	// Check buffer alarm
	IF fbMFCS_Channel[E_MFCS_Channel.AM].M_BufferLevelAlarm() THEN	
		// Set error
		F_SetError(	
			ErrorType	:= E_ErrorType.ERROR,
			ErrorParam	:= '',
			ErrorMsg	:= E_ErrorConv.AM_BUFFER_OVERFLOW,
			ErrorData	:= SubsystemData.ErrorData.ErrorDataSet[7]);
			
	// Check buffer warning
	ELSIF fbMFCS_Channel[E_MFCS_Channel.AM].M_BufferLevelWarning() AND
	      SubsystemData.ErrorData.ErrorDataSet[7].ErrorType <> E_ErrorType.ERROR THEN
		// Set error
		F_SetError(	
			ErrorType	:= E_ErrorType.WARNING,
			ErrorParam	:= '',
			ErrorMsg	:= E_ErrorConv.AM_BUFFER_OVERFLOW,
			ErrorData	:= SubsystemData.ErrorData.ErrorDataSet[7]);
	ELSE
		// Reset error
		F_ResetError(Reset := TRUE, ErrorData := SubsystemData.ErrorData.ErrorDataSet[7]);
		
	END_IF
ELSE
	// Reset error
	F_ResetError(Reset := TRUE, ErrorData := SubsystemData.ErrorData.ErrorDataSet[6]);
	F_ResetError(Reset := TRUE, ErrorData := SubsystemData.ErrorData.ErrorDataSet[7]);
	
	// Reset command to stop
	StopAllGroups := FALSE;
END_IF

(**************************************************************************************
   SPOC Connection
***************************************************************************************)
// If SPOC is configured
IF Settings.SPOC_Exists THEN
	
	// If SPOC is not connected
	IF NOT fbMFCS_Channel[E_MFCS_Channel.SPOC].M_IsConnected() THEN
		// Set error
		F_SetError(	
			ErrorType	:= E_ErrorType.ERROR,
			ErrorParam	:= '',
			ErrorMsg	:= E_ErrorConv.CONNECTION_ERROR_TO_SPOC,
			ErrorData	:= SubsystemData.ErrorData.ErrorDataSet[8]);
	ELSE
		// Reset error
		F_ResetError(Reset := TRUE,ErrorData := SubsystemData.ErrorData.ErrorDataSet[8]);
	END_IF
ELSE
	// Reset error
	F_ResetError(Reset := TRUE,ErrorData := SubsystemData.ErrorData.ErrorDataSet[8]);
END_IF
END_ACTION

ACTION A_OutputMapping:
(**************************************************************************************
 * 	NAME		A_OutputMapping
 * 	FUNCTION	Output mapping
 **************************************************************************************)

 
 
(**************************************************************************************************************
   Outputs
***************************************************************************************************************)
SubsystemInterface.Out.MasterSpeed := SubsystemInterface.In.MasterSpeed;
END_ACTION

ACTION A_SlaveDeviceSupervision:
(**************************************************************************************
 * 	NAME		A_SlaveDeviceSupervision
 * 	FUNCTION	Check connected EtherCAT Slaves for diagnostic reasons
 *
 *				0x___1 = Slave in 'INIT' state
 *	 			0x___2 = Slave in 'PREOP' state
 *				0x___3 = Slave in 'BOOT' state
 *				0x___4 = Slave in 'SAFEOP' state
 *				0x___8 = Slave in 'OP' state
 *				0x001_ = Slave signals error
 *				0x002_ = Invalid vendorId, productCode... read
 *				0x004_ = Initialization error occurred
 *				0x008_ = Slave disabled
 *				0x010_ = Slave not present
 *				0x020_ = Slave signals link error
 *				0x040_ = Slave signals missing link
 *				0x080_ = Slave signals unexpected link
 *				0x100_ = Communication port A
 *				0x200_ = Communication port B
 *				0x400_ = Communication port C
 *				0x800_ = Communication port D
 *
 **************************************************************************************)
 
// Check all device slaves 
FOR Idx := 1 TO NUMBERS_OF_ETHERCAT_SLAVE_DIAG DO
	// If state is >16 and state has changed
	IF Inputs.DeviceState[Idx] >= 16 AND Inputs.DeviceState[Idx] <> EtherCatSupervision[Idx].DeviceState THEN
		// Update event list
		EtherCatSupervision[Idx].EventDateTime 			:= TimeStampDT;
		EtherCatSupervision[Idx].Error 					:= TRUE;
		EtherCatSupervision[Idx].LastDeviceState		:= EtherCatSupervision[Idx].DeviceState;
		EtherCatSupervision[Idx].DeviceState			:= Inputs.DeviceState[Idx];
		
		// Print debug
		DebugMsg := CONCAT('EtherCAT-Device Error, Device: ', INT_TO_STRING(Idx));
		DebugMsg := CONCAT(DebugMsg, ' Last Device state: ');
		DebugMsg := CONCAT(DebugMsg, UINT_TO_STRING(EtherCatSupervision[Idx].LastDeviceState));
		DebugMsg := CONCAT(DebugMsg, ' Device state: ');
		DebugMsg := CONCAT(DebugMsg, UINT_TO_STRING(EtherCatSupervision[Idx].DeviceState));
		DebugMsg := CONCAT(DebugMsg, ' Active: ');
		DebugMsg := CONCAT(DebugMsg, BOOL_TO_STRING(EtherCatSupervision[Idx].Error));
		fbDebugMsg.M_SendInfoMsg(DebugMsg);
		
	// If no error is active - update table
	ELSIF Inputs.DeviceState[Idx] <> EtherCatSupervision[Idx].DeviceState THEN
		// Reset table
		EtherCatSupervision[Idx].LastDeviceState		:= EtherCatSupervision[Idx].DeviceState;
		EtherCatSupervision[Idx].DeviceState			:= Inputs.DeviceState[Idx];
		EtherCatSupervision[Idx].Error	 				:= FALSE;
		
		// Print debug
		DebugMsg := CONCAT('EtherCAT-Device Error, Device: ', INT_TO_STRING(Idx));
		DebugMsg := CONCAT(DebugMsg, ' Last Device state: ');
		DebugMsg := CONCAT(DebugMsg, UINT_TO_STRING(EtherCatSupervision[Idx].LastDeviceState));
		DebugMsg := CONCAT(DebugMsg, ' Device state: ');
		DebugMsg := CONCAT(DebugMsg, UINT_TO_STRING(EtherCatSupervision[Idx].DeviceState));
		DebugMsg := CONCAT(DebugMsg, ' Active: ');
		DebugMsg := CONCAT(DebugMsg, BOOL_TO_STRING(EtherCatSupervision[Idx].Error));
		fbDebugMsg.M_SendInfoMsg(DebugMsg);
	END_IF
END_FOR
END_ACTION

ACTION A_StateControl:
(**************************************************************************************
 * 	NAME		A_StateControl
 * 	FUNCTION	State control 
 **************************************************************************************)

// Update system state
SubSystemData.OperationState.Info.SystemReady := SubSystemData.OperationState.eState = E_PositionState.STARTED;
 
// Group states
CASE SubSystemData.OperationState.eState OF
	(*******************************************************************************
	  Unknown State 
	********************************************************************************)
	E_PositionState.UNKNOWN:
		// Subsystem default state
		SubSystemData.OperationState.eLastState := SubSystemData.OperationState.eState;
		SubSystemData.OperationState.eState 	:= E_PositionState.STOPPED;

	(*******************************************************************************
	  Stopped
	********************************************************************************)
	E_PositionState.STOPPED:
		IF SubSystemData.ErrorData.ErrorDataSet[7].ErrorType <> E_ErrorType.ERROR AND
		   SubSystemData.ErrorData.ErrorDataSet[7].ErrorType <> E_ErrorType.WARNING THEN
		   
		   // Change state "Starting"
			SubSystemData.OperationState.eLastState := SubSystemData.OperationState.eState;
			SubSystemData.OperationState.eState := E_PositionState.STARTING;
		
			// Send status report
			ITC.Commands.StatusReport := TRUE;
		END_IF
		
	(*******************************************************************************
	  Stopping
	********************************************************************************)
	E_PositionState.STOPPING:
		fbStoppingDelayTimer(IN := TRUE, PT := Settings.tDelayStopping);
	
		// If no "AM_Buffer" error is pending
		IF SubSystemData.ErrorData.ErrorDataSet[7].ErrorType = E_ErrorType.ERROR OR 
		   fbStoppingDelayTimer.Q THEN
		   
			// Change state "Stopped"
			SubSystemData.OperationState.eLastState := SubSystemData.OperationState.eState;
			SubSystemData.OperationState.eState := E_PositionState.STOPPED;
		
			// Send status report
			ITC.Commands.StatusReport := TRUE;
			
			fbStoppingDelayTimer(IN := FALSE);
			
		// If no "AM_BUffer" warning is pending
		ELSIF SubSystemData.ErrorData.ErrorDataSet[7].ErrorType = E_ErrorType.WARNING THEN
			// Wait
			;
		ELSE
			// Start again
			SubSystemData.OperationState.eLastState := SubSystemData.OperationState.eState;
			SubSystemData.OperationState.eState := E_PositionState.STARTING;
		
			// Send status report
			ITC.Commands.StatusReport := TRUE;
		END_IF

	(*******************************************************************************
	  Starting
	********************************************************************************)
	E_PositionState.STARTING:
		// If no "AM_Buffer" error/warning is pending
		IF SubSystemData.ErrorData.ErrorDataSet[7].ErrorType = E_ErrorType.ERROR OR
   		   SubSystemData.ErrorData.ErrorDataSet[7].ErrorType = E_ErrorType.WARNING THEN
			// Change state "Stopped"
			SubSystemData.OperationState.eLastState := SubSystemData.OperationState.eState;
			SubSystemData.OperationState.eState := E_PositionState.STOPPED;
		
			// Send status report
			ITC.Commands.StatusReport := TRUE;
			
		ELSIF fbStartUpDelayTimer.Q THEN
			// Change state "Started"
			SubSystemData.OperationState.eLastState := SubSystemData.OperationState.eState;
			SubSystemData.OperationState.eState := E_PositionState.STARTED;
		
			// Send status report
			ITC.Commands.StatusReport := TRUE;
		END_IF
		
	(*******************************************************************************
	  Started (Online/active/running)
	********************************************************************************)
	E_PositionState.STARTED:
	
		// If no "AM_Buffer" error is pending
		IF SubSystemData.ErrorData.ErrorDataSet[7].ErrorType = E_ErrorType.ERROR OR
		   NOT fbStartUpDelayTimer.Q THEN
			// Change state "Stopped"
			SubSystemData.OperationState.eLastState := SubSystemData.OperationState.eState;
			SubSystemData.OperationState.eState := E_PositionState.STOPPED;
			// Send status report
			ITC.Commands.StatusReport := TRUE;
			
		// If no "AM_BUffer" warning is pending
		ELSIF SubSystemData.ErrorData.ErrorDataSet[7].ErrorType = E_ErrorType.WARNING THEN
			// Change state "Stopping"
			SubSystemData.OperationState.eLastState := SubSystemData.OperationState.eState;
			SubSystemData.OperationState.eState := E_PositionState.STOPPING;
		
			// Send status report
			ITC.Commands.StatusReport := TRUE;
			fbStoppingDelayTimer(IN := FALSE);
		END_IF
		
(********************************************************************************
	Error case
*********************************************************************************)
ELSE
	// Programming error
	DebugMsg := CONCAT(	'Programming error - Invalid state: ', INT_TO_STRING(SubSystemData.OperationState.eState));
	fbDebugMsg.M_SendErrorMsg(DebugMsg);
END_CASE
END_ACTION

ACTION A_UpdateSystemTime:
(**************************************************************************************
 * 	NAME		A_UpdateSystemTime
 * 	FUNCTION	Updates the SystemTime of the IPC
 *
 **************************************************************************************)
 
// Check if it is more than 24h ago since the last synchronization 
IF TimeStampDT - LastSystemTimeUpdate > Settings.MinTimeSync AND 
   Settings.EnableTimeSync AND
   NOT UpdateSystemTime THEN

		// Update in progress
		UpdateSystemTime := TRUE;

		// Request time synchronization
		ITC.Commands.RequestTimeUpdate := TRUE;
		
		// Reset timer
		fbTimeReqReset(IN := FALSE);
END_IF


// If an update was requested
IF UpdateSystemTime THEN
	// Start timer to reset request
	fbTimeReqReset(IN := TRUE, PT:= Settings.tRequestReset);
	
	// If no telegram was received in a certain time
	IF fbTimeReqReset.Q THEN
		// Reset request to resend a new one
		UpdateSystemTime := FALSE;
		
		// Reset timer
		fbTimeReqReset(IN := FALSE);

		// debug
		DebugMsg := 'No time synchronization telegram received. ';
		DebugMsg := CONCAT(	DebugMsg, 'Current system time: ');
		DebugMsg := CONCAT(	DebugMsg, DT_TO_STRING(TimeStampDT));
		fbDebugMsg.M_SendWarningMsg(DebugMsg);		
	END_IF
END_IF


// A synchronization telegram was received 
IF ITC.Commands.UpdateSystemTime THEN
	// Call time sync
	fbUpdateSystemTime(START := FALSE);

	// If no sync command is active
	IF NOT TimeSyncActive THEN
		// Call time sync
		fbUpdateSystemTime(
			START 	:= TRUE,
			TIMESTR := STRING_TO_SYSTEMTIME(SubsystemBase.TimeValue));

		// Sync active
		TimeSyncActive := TRUE;
	
	ELSIF NOT fbUpdateSystemTime.BUSY THEN
		// Update finished
		UpdateSystemTime := FALSE;
		ITC.Commands.UpdateSystemTime := FALSE;
		TimeSyncActive 	:= FALSE;
		
		// Update new time stamp
		LastSystemTimeUpdate := TimeStampDT;
		
		// debug
		DebugMsg := CONCAT(	'Time sync done - New: ',SubsystemBase.TimeValue);
		DebugMsg := CONCAT(	DebugMsg, ' Old: ');
		DebugMsg := CONCAT(	DebugMsg, DT_TO_STRING(TimeStampDT));
		fbDebugMsg.M_SendInfoMsg(DebugMsg);
	END_IF
END_IF
END_ACTION

END_FUNCTION_BLOCK

// ---- 20_Product/10_BCF/11_Conv/15_Subsystem/FB_SubsystemConv.TcPOU
FUNCTION_BLOCK FB_SubsystemConv EXTENDS FB_BaseObject
(**************************************************************************************
 * 	Application		:	BoxControl Framework
 *	Revision		:	$Revision: 404529 $
 *	Revision date	:	$Date: 2020-11-19 15:59:09 +0100 (tor, 19 nov 2020) $
 *	Last changed by	:	$Author: b7bolm $
 *	URL				:	$URL: http://almscdc.swisslog.com/repo/SWPD/Development/BoxControlFramework/20_Release/trunk/01_Software/BCF/BCF/JumpStart/20_Product/10_App/15_Subsystem/10_Lib/10_Conv/FB_SubsystemConv.TcPOU $
 *
 *	Purpose			:	Main subsystem
 *
 * ------------------------------------------------------------------------------------
 *	Copyright Swisslog [IP AG], Switzerland. All rights reserved.
 * 
 * ------------------------------------------------------------------------------------
 *	
 * 	Revision History: 
 *
 * 	VERSION			DATE			INITIALS			DESCRIPTION
 *	0.1				01.01.2001		swl					Example
 *
 **************************************************************************************)
VAR_INPUT
	ConfigSubsystem				: ST_CFG_Subsystem; // Configuration 
END_VAR

VAR
	SubsystemBase				: ST_SubsystemBase; // Subsystem base	
END_VAR

VAR PERSISTENT
	ITC							: ST_ITC_Subsystem; // Internal ITC
	SubsystemData				: ST_SubsystemData; // Subsystem data
	SubsystemInterface			: ST_SubsystemInterface; // Interface to the Subsystem 
	SettingsSubsystem			: ST_CFG_Subsystem; // Settings
END_VAR

(**************************************************************************************************************
   Base Subsystem - Body is never called!
***************************************************************************************************************)
;

METHOD M_InitControl : BOOL
(**************************************************************************************
 * 	Application		:	BoxControl Framework
 *	Revision		:	$Revision: 404529 $
 *	Revision date	:	$Date: 2020-11-19 15:59:09 +0100 (tor, 19 nov 2020) $
 *	Last changed by	:	$Author: b7bolm $
 *	URL				:	$URL: http://almscdc.swisslog.com/repo/SWPD/Development/BoxControlFramework/20_Release/trunk/01_Software/BCF/BCF/JumpStart/20_Product/10_App/15_Subsystem/10_Lib/10_Conv/FB_SubsystemConv.TcPOU $
 *
 *	Purpose			:	Control initialization sequence
 *
 * ------------------------------------------------------------------------------------
 *	Copyright Swisslog [IP AG], Switzerland. All rights reserved.
 * 
 * ------------------------------------------------------------------------------------
 *	
 * 	Revision History: 
 *
 * 	VERSION			DATE			INITIALS			DESCRIPTION
 *	0.1				01.01.2001		swl					Example
 *
 **************************************************************************************)

// If groupwise initialization is enabled
IF SettingsSubsystem.MaxInitCallsPerCycle <> 0 THEN
	// If the subsystem is started
	IF SubsystemData.OperationState.eState = E_PositionState.STARTED THEN
		(*
		In order to control the PLC load due to initialization, 
		all positions will be initialized in groups.
		
		Order:
			1. Group
			2. Element
			3. Function
		*)
		IF SubsystemBase.eLimitGroupNumber < E_GroupNumber.G_END_GROUP THEN
		
			IF SubsystemBase.eLimitGroupNumber + SettingsSubsystem.MaxInitCallsPerCycle > E_GroupNumber.G_END_GROUP THEN
				SubsystemBase.eLimitGroupNumber := E_GroupNumber.G_END_GROUP;
				SubsystemData.OperationState.InitRelease.eLimitGroup := E_GroupNumber.G_END_GROUP;
			ELSE
				SubsystemBase.eLimitGroupNumber :=  SubsystemBase.eLimitGroupNumber + SettingsSubsystem.MaxInitCallsPerCycle;
				SubsystemData.OperationState.InitRelease.eLimitGroup := SubsystemBase.eLimitGroupNumber;
			END_IF
		ELSIF SubsystemBase.eLimitElementNumber < E_ElementNumber.E_END_ELEMENT THEN
		
			IF SubsystemBase.eLimitElementNumber + SettingsSubsystem.MaxInitCallsPerCycle > E_ElementNumber.E_END_ELEMENT THEN
				SubsystemBase.eLimitElementNumber := E_ElementNumber.E_END_ELEMENT;
				SubsystemData.OperationState.InitRelease.eLimitElementNumber := SubsystemBase.eLimitElementNumber;
			ELSE
				SubsystemBase.eLimitElementNumber :=  SubsystemBase.eLimitElementNumber + SettingsSubsystem.MaxInitCallsPerCycle;
				SubsystemData.OperationState.InitRelease.eLimitElementNumber := SubsystemBase.eLimitElementNumber;
			END_IF
		ELSIF SubsystemBase.eLimitFunctionNumber < E_FunctionNumber.F_END_FUNCTION THEN
		
			IF SubsystemBase.eLimitFunctionNumber + SettingsSubsystem.MaxInitCallsPerCycle > E_FunctionNumber.F_END_FUNCTION THEN
				SubsystemBase.eLimitFunctionNumber := E_FunctionNumber.F_END_FUNCTION;
				SubsystemData.OperationState.InitRelease.eLimitFunctionNumber := SubsystemBase.eLimitFunctionNumber;
			ELSE
				SubsystemBase.eLimitFunctionNumber :=  SubsystemBase.eLimitFunctionNumber + SettingsSubsystem.MaxInitCallsPerCycle;
				SubsystemData.OperationState.InitRelease.eLimitFunctionNumber := SubsystemBase.eLimitFunctionNumber;
			END_IF
		END_IF
	ELSE
		SubsystemBase.eLimitFunctionNumber := E_FunctionNumber.F_BEGIN_FUNCTION;
		SubsystemBase.eLimitElementNumber := E_ElementNumber.E_BEGIN_ELEMENT;
		SubsystemBase.eLimitGroupNumber := E_GroupNumber.G_BEGIN_GROUP;
	END_IF
ELSE
	SubsystemBase.eLimitFunctionNumber := E_FunctionNumber.F_END_FUNCTION;
	SubsystemBase.eLimitElementNumber := E_ElementNumber.E_END_ELEMENT;
	SubsystemBase.eLimitGroupNumber := E_GroupNumber.G_END_GROUP;
	SubsystemData.OperationState.InitRelease.eLimitGroup := SubsystemBase.eLimitGroupNumber;
	SubsystemData.OperationState.InitRelease.eLimitElementNumber := SubsystemBase.eLimitElementNumber;
	SubsystemData.OperationState.InitRelease.eLimitFunctionNumber := SubsystemBase.eLimitFunctionNumber;
END_IF
END_METHOD

METHOD M_InitSubsystem : BOOL
(**************************************************************************************
 * 	Application		:	BoxControl Framework
 *	Revision		:	$Revision: 404529 $
 *	Revision date	:	$Date: 2020-11-19 15:59:09 +0100 (tor, 19 nov 2020) $
 *	Last changed by	:	$Author: b7bolm $
 *	URL				:	$URL: http://almscdc.swisslog.com/repo/SWPD/Development/BoxControlFramework/20_Release/trunk/01_Software/BCF/BCF/JumpStart/20_Product/10_App/15_Subsystem/10_Lib/10_Conv/FB_SubsystemConv.TcPOU $
 *
 *	Purpose			:	Initialize SubSystem
 *
 * ------------------------------------------------------------------------------------
 *	Copyright Swisslog [IP AG], Switzerland. All rights reserved.
 * 
 * ------------------------------------------------------------------------------------
 *	
 * 	Revision History: 
 *
 * 	VERSION			DATE			INITIALS			DESCRIPTION
 *	0.1				01.01.2001		swl					Example
 *
 **************************************************************************************)
  VAR_INPUT
	 mReset		: BOOL; // Force initialization
 END_VAR
 VAR
	 mName		: T_MaxString; // Name with alpha numeric signs only
 END_VAR
// If the init command was an external command
IF mReset THEN
	// Inform the bottom subsystem to initialize
	SubSystemData.Init := FALSE;
	// Reset values and load config
	M_PreInit();
ELSE
	// Load basic configuration to settings
	SettingsSubsystem := ConfigSubsystem;
	
	// Remove non alpha numeric signs
	mName := F_ReduceToAlphaNumeric(InputString := SettingsSubsystem.SubsystemName);

	// Update Registry reference with HashCode
	SubsystemRegistry.HashCode := F_CreateHashCode(mName);
	
	// Update Registry reference with name
	SubsystemRegistry.SubsystemName := SettingsSubsystem.SubsystemName;
	
	// Base subsystem initialized
	M_InitSubsystem := TRUE;
END_IF
END_METHOD

METHOD M_ITC_ProcessMsg : BOOL
(**************************************************************************************
 * 	Application		:	BoxControl Framework
 *	Revision		:	$Revision: 404529 $
 *	Revision date	:	$Date: 2020-11-19 15:59:09 +0100 (tor, 19 nov 2020) $
 *	Last changed by	:	$Author: b7bolm $
 *	URL				:	$URL: http://almscdc.swisslog.com/repo/SWPD/Development/BoxControlFramework/20_Release/trunk/01_Software/BCF/BCF/JumpStart/20_Product/10_App/15_Subsystem/10_Lib/10_Conv/FB_SubsystemConv.TcPOU $
 *
 *	Purpose			:	Handle incoming group ITC messages.
 *
 * ------------------------------------------------------------------------------------
 *	Copyright Swisslog [IP AG], Switzerland. All rights reserved.
 * 
 * ------------------------------------------------------------------------------------
 *	
 * 	Revision History: 
 *
 * 	VERSION			DATE			INITIALS			DESCRIPTION
 *	0.1				01.01.2001		swl					Example
 *
 **************************************************************************************)
VAR_INPUT
	meChannelSrc		: E_MFCS_CHANNEL; // Number of the source 
	mMsgType			: INT; // Message type
	mpData				: PVOID; // Data  pointer 
	mLen				: UDINT; // Data length
END_VAR
// Initialize
M_ITC_ProcessMsg := TRUE;

// Validate inputs
IF mpData > 0 AND
   mLen > 0 THEN
	// Map enum
	SubsystemBase.eMsgType := mMsgType;

	// Validate message type
	CASE SubsystemBase.eMsgType OF
		(*******************************************************************************
		  Status request message
		********************************************************************************)
		E_ITC_MsgTypeConv.SUBSYSTEM_STATUS_REQUEST:		
			M_ITC_SSQ(meChannelSrc := meChannelSrc, mpData := mpData, mLen := mLen);
			
		(*******************************************************************************
		  Control request message
		********************************************************************************)
		E_ITC_MsgTypeConv.SUBSYSTEM_CONTROL_REQUEST:
			M_ITC_SCQ(meChannelSrc := meChannelSrc, mpData := mpData, mLen := mLen);

						
		(*******************************************************************************
		  Data Aquisition Request 
		********************************************************************************)
		E_ITC_MsgTypeConv.DATA_ACQUISITION_REQUEST:
			M_ITC_DAQ(meChannelSrc := meChannelSrc, mpData := mpData, mLen := mLen);
		(*******************************************************************************
		  Gathered Data Request 
		********************************************************************************)
		E_ITC_MsgTypeConv.GATHERED_DATA_REQUEST:
			M_ITC_GDQ(meChannelSrc := meChannelSrc, mpData := mpData, mLen := mLen);
			
		(*******************************************************************************
		  Visualization information request
		********************************************************************************)			
		E_ITC_MsgTypeConv.VISUALIZATION_INFORMATION_REQUEST:
			M_ITC_VIQ(meChannelSrc := meChannelSrc, mpData := mpData, mLen := mLen);
				

	ELSE
		// Unknown ITC message type received
		DebugMsg := CONCAT('M_ITC_HandleBufferMessages - Unknown message type received: ', INT_TO_STRING(mMsgType));
		fbDebugMsg.M_SendErrorMsg(mMessage := DebugMsg);
	END_CASE
END_IF
END_METHOD

METHOD M_ITC_ProcessOut : BOOL
(**************************************************************************************
 * 	Application		:	BoxControl Framework
 *	Revision		:	$Revision: 404529 $
 *	Revision date	:	$Date: 2020-11-19 15:59:09 +0100 (tor, 19 nov 2020) $
 *	Last changed by	:	$Author: b7bolm $
 *	URL				:	$URL: http://almscdc.swisslog.com/repo/SWPD/Development/BoxControlFramework/20_Release/trunk/01_Software/BCF/BCF/JumpStart/20_Product/10_App/15_Subsystem/10_Lib/10_Conv/FB_SubsystemConv.TcPOU $
 *
 *	Purpose			:	Subsystem ITC out interface
 *						Handles internally set ITC commands.
 *
 * ------------------------------------------------------------------------------------
 *	Copyright Swisslog [IP AG], Switzerland. All rights reserved.
 * 
 * ------------------------------------------------------------------------------------
 *	
 * 	Revision History: 
 *
 * 	VERSION			DATE			INITIALS			DESCRIPTION
 *	0.1				01.01.2001		swl					Example
 *
 **************************************************************************************)
VAR
	mErrorData	 		: ST_SubsystemErrorStruct; // Error data
	mNoError			: BOOL; // No error during processing
	mSSR				: ST_ITC_SSR; // ITC struct
	mSCR				: ST_ITC_SCR; // ITC struct
	mNumberOfZones		: INT; // Number of zones
	mZoneIdx			: INT; // Zone index
END_VAR

(*******************************************************************************
	Status Report : System restart
********************************************************************************)
// If a system restart info request is active
IF ITC.Commands.SystemRestartInfo THEN
	// Get error data
	mErrorData := SubsystemData.ErrorData;
	
	mNoError := F_ITC_SendSSR(
					eChannelSrc		:= 0, 
					SubsystemName	:= F_ReduceToAlphaNumeric(SettingsSubsystem.SubsystemName), 
					eMode			:= SubsystemData.OperationState.eMode, 
					eState			:= SubsystemData.OperationState.eState, 
					eSystemInfo		:= E_SystemInfo.RESTARTED, 
					eErrorState		:= mErrorData.ErrorState, 
					eErrorCode		:= mErrorData.Error.ErrorCode.Conv, 
					eErrorType		:= mErrorData.Error.ErrorType, 
					ErrorInformation:= mErrorData.Error.ErrorParam, 
					Variable		:= ITC.Variable, 
					eReturnCode		:= E_ErrorConv.NO_ERROR_CODE);

	// If sending was successfull
	IF mNoError THEN
		// Reset flag
		ITC.Commands.SystemRestartInfo := FALSE;
	ELSE
		// Sending failed
		DebugMsg := 'M_ITC_ProcessOut - Forwarding system restart to ITC manager failed.';
		fbDebugMsg.M_SendErrorMsg(mMessage := DebugMsg);
	END_IF
END_IF

(*******************************************************************************
	Status Report : No error
********************************************************************************)
// If an error is gone, send status report
IF ITC.Commands.NoErrorReport THEN

	// Get error data
	mErrorData := SubsystemData.ErrorData;
	
	mNoError := F_ITC_SendSSR(
					eChannelSrc		:= 0, 
					SubsystemName	:= F_ReduceToAlphaNumeric(SettingsSubsystem.SubsystemName), 
					eMode			:= SubsystemData.OperationState.eMode, 
					eState			:= SubsystemData.OperationState.eState, 
					eSystemInfo		:= E_SystemInfo.NO_INFO, 
					eErrorState		:= E_ErrorState.OPERATIONAL, 
					eErrorCode		:= E_ErrorConv.NO_ERROR_CODE, 
					eErrorType		:= E_ErrorType.NO_ERROR_PENDING, 
					ErrorInformation:= '', 
					Variable		:= ITC.Variable, 
					eReturnCode		:= E_ErrorConv.NO_ERROR_CODE);

	// If sending was successfull
	IF mNoError THEN
		// Reset flag
		ITC.Commands.NoErrorReport := FALSE;
	ELSE
		// Sending failed
		DebugMsg := 'M_ITC_ProcessOut - Forwarding "No error" status report to ITC manager failed.';
		fbDebugMsg.M_SendErrorMsg(mMessage := DebugMsg);
	END_IF
END_IF

(*******************************************************************************
	Status Report : Time request
********************************************************************************)
// If a system restart info request is active
IF ITC.Commands.RequestTimeUpdate THEN

	// Get error data
	mErrorData := SubsystemData.ErrorData;
	
	mNoError := F_ITC_SendSSR(
					eChannelSrc		:= 0, 
					SubsystemName	:= F_ReduceToAlphaNumeric(SettingsSubsystem.SubsystemName), 
					eMode			:= SubsystemData.OperationState.eMode, 
					eState			:= SubsystemData.OperationState.eState, 
					eSystemInfo		:= E_SystemInfo.TIME_UPDATE_REQUIRED, 
					eErrorState		:= mErrorData.ErrorState, 
					eErrorCode		:= mErrorData.Error.ErrorCode.Conv, 
					eErrorType		:= mErrorData.Error.ErrorType, 
					ErrorInformation:= mErrorData.Error.ErrorParam, 
					Variable		:= ITC.Variable, 
					eReturnCode		:= E_ErrorConv.NO_ERROR_CODE);
					
					
	// If sending was successfull
	IF mNoError THEN
		// Reset flag
		ITC.Commands.RequestTimeUpdate := FALSE;
	ELSE
		// Sending failed
		DebugMsg := 'M_ITC_ProcessOut - Forwarding request time update to ITC manager failed.';
		fbDebugMsg.M_SendErrorMsg(mMessage := DebugMsg);
	END_IF
END_IF

(*******************************************************************************
	Status Report 
********************************************************************************)
// If a time request request is active
IF ITC.Commands.StatusReport THEN

	// Get error data
	mErrorData := SubsystemData.ErrorData;

	mNoError := F_ITC_SendSSR(
					eChannelSrc		:= 0, 
					SubsystemName	:= F_ReduceToAlphaNumeric(SettingsSubsystem.SubsystemName), 
					eMode			:= SubsystemData.OperationState.eMode, 
					eState			:= SubsystemData.OperationState.eState, 
					eSystemInfo		:= E_SystemInfo.NO_INFO, 
					eErrorState		:= mErrorData.ErrorState, 
					eErrorCode		:= mErrorData.Error.ErrorCode.Conv, 
					eErrorType		:= mErrorData.Error.ErrorType, 
					ErrorInformation:= mErrorData.Error.ErrorParam, 
					Variable		:= ITC.Variable, 
					eReturnCode		:= E_ErrorConv.NO_ERROR_CODE);

	// If sending was successfull
	IF mNoError THEN
		// Reset flag
		ITC.Commands.StatusReport := FALSE;
	ELSE
		// Sending failed
		DebugMsg := 'M_ITC_ProcessOut - Forwarding status report to ITC manager failed.';
		fbDebugMsg.M_SendErrorMsg(mMessage := DebugMsg);
	END_IF
END_IF

(*******************************************************************************
	Control Report 
********************************************************************************)
// If a control report msg request is active
IF ITC.Commands.ControlReport THEN

	mNoError := F_ITC_SendSCR(
					eChannelSrc		:= 0, 
					SubsystemName	:= F_ReduceToAlphaNumeric(SettingsSubsystem.SubsystemName), 
					Code			:= 0, 
					Variable		:= ITC.Variable, 
					eReturnCode		:= E_ErrorConv.NO_ERROR_CODE);

	// If sending was successfull
	IF mNoError THEN
		// Reset flag
		ITC.Commands.ControlReport := FALSE;
	ELSE
		// Sending failed
		DebugMsg := 'M_ITC_ProcessOut - Forwarding control report to ITC manager failed.';
		fbDebugMsg.M_SendErrorMsg(mMessage := DebugMsg);
	END_IF
END_IF

(*******************************************************************************
	Command to send update of the whole system
********************************************************************************)
// If a Update all group and postion msg request is active
IF ITC.Commands.UpdateAllGroupsAndPositions THEN
	(*
	A full system update needs a lot of system ressources, 
	therefore the request is separated in several cycles instead
	of sending all telegrams in one cycle.
	*)

	// Forward request to all groups in the registry
	IF SubsystemBase.eUpdateGroupNumber > E_GroupNumber.G_BEGIN_GROUP  AND 
	   SubsystemBase.eUpdateGroupNumber < E_GroupNumber.G_END_GROUP THEN
		// Forward request
		SubsystemBase.GSQ.Position := F_ReduceToAlphaNumeric(GroupRegistry[SubsystemBase.eUpdateGroupNumber].GroupName);

		System.fbITC_Manager.M_AddData(
			meChannelSrc := SubsystemBase.UpdateChannelSrc,
			mMsgType 	 := E_ITC_MsgTypeConv.GROUP_STATUS_REQUEST,
			mpData		 := ADR(SubsystemBase.GSQ),
			mLen		 := SIZEOF(SubsystemBase.GSQ));
		
		// Increment index or terminate sending group status	
		IF SubsystemBase.eUpdateGroupNumber < E_GroupNumber.G_END_GROUP THEN 
			SubsystemBase.eUpdateGroupNumber := SubsystemBase.eUpdateGroupNumber + 1;
		END_IF	
	ELSE
		SubsystemBase.UpdateGroupDone := TRUE;
	END_IF
	
	// Forward request to all elements in the registry
	IF SubsystemBase.eUpdateElementNumber > E_ElementNumber.E_BEGIN_ELEMENT  AND 
	   SubsystemBase.eUpdateElementNumber < E_ElementNumber.E_END_ELEMENT THEN	
		// Forward request
		SubsystemBase.ESQ.Position := F_ReduceToAlphaNumeric(ElementRegistry[SubsystemBase.eUpdateElementNumber].ElementName);
		
		System.fbITC_Manager.M_AddData(
			meChannelSrc := SubsystemBase.UpdateChannelSrc,
			mMsgType 	 := E_ITC_MsgTypeConv.Element_STATUS_REQUEST,
			mpData		 := ADR(SubsystemBase.ESQ),
			mLen		 := SIZEOF(SubsystemBase.ESQ));
			
		// Increment index or terminate sending element status
		IF SubsystemBase.eUpdateElementNumber < E_ElementNumber.E_END_ELEMENT THEN 
			SubsystemBase.eUpdateElementNumber := SubsystemBase.eUpdateElementNumber + 1;
		END_IF			
	ELSE
		SubsystemBase.UpdateElementDone := TRUE;
	END_IF
	
	// Forward request to all functions and zones in the registry
	IF SubsystemBase.eUpdateFunctionNumber > E_FunctionNumber.F_BEGIN_FUNCTION  AND 
	   SubsystemBase.eUpdateFunctionNumber < E_FunctionNumber.F_END_FUNCTION THEN	
		// Forward request
		SubsystemBase.FSQ.Position := F_ReduceToAlphaNumeric(FunctionRegistry[SubsystemBase.eUpdateFunctionNumber].FunctionName);

		System.fbITC_Manager.M_AddData(
			meChannelSrc := SubsystemBase.UpdateChannelSrc,
			mMsgType 	 := E_ITC_MsgTypeConv.FUNCTION_STATUS_REQUEST,
			mpData		 := ADR(SubsystemBase.FSQ),
			mLen		 := SIZEOF(SubsystemBase.FSQ));
	
		// Get function settings
		mNumberOfZones := F_GetNumberOfZones(eFunctionNumber := SubsystemBase.eUpdateFunctionNumber);

		// Go through all configured zones
		FOR mZoneIdx := 1 TO mNumberOfZones DO
			SubsystemBase.FSQ.Position := F_ReduceToAlphaNumeric(FunctionRegistry[SubsystemBase.eUpdateFunctionNumber].Zone[mZoneIdx].ZoneName);
			
			System.fbITC_Manager.M_AddData(
				meChannelSrc := SubsystemBase.UpdateChannelSrc,
				mMsgType 	 := E_ITC_MsgTypeConv.FUNCTION_STATUS_REQUEST,
				mpData		 := ADR(SubsystemBase.FSQ),
				mlen		 := SIZEOF(SubsystemBase.FSQ));
		END_FOR
		// Increment index or terminate function status
		IF SubsystemBase.eUpdateFunctionNumber < E_FunctionNumber.F_END_FUNCTION THEN 
			SubsystemBase.eUpdateFunctionNumber := SubsystemBase.eUpdateFunctionNumber + 1;
		END_IF			
	ELSE
		SubsystemBase.UpdateFunctionDone := TRUE;		
	END_IF

	// If all status are reported 
	IF SubsystemBase.UpdateGroupDone AND 
	   SubsystemBase.UpdateElementDone AND 
       SubsystemBase.UpdateFunctionDone THEN
		// Terminate reporting
		SubsystemBase.UpdateGroupDone := FALSE;
		SubsystemBase.UpdateElementDone := FALSE;
		SubsystemBase.UpdateFunctionDone := FALSE;		
		ITC.Commands.UpdateAllGroupsAndPositions := FALSE;
	END_IF
END_IF
END_METHOD

METHOD PRIVATE M_ITC_SCQ : BOOL
VAR_INPUT
	meChannelSrc		: E_MFCS_CHANNEL; // Number of the source 
	mpData				: PVOID; // Data  pointer 
	mLen				: UDINT; // Data length
END_VAR
// Map data
F_BlockCopy(
	pSrc:= mpData, 
	LenSrc:= mLen, 
	pDest:= ADR(SubsystemBase.SCQ), 
	LenDest:= SIZEOF(SubsystemBase.SCQ));
	
// Validate control code
CASE SubsystemBase.SCQ.Code OF
	(*******************************************************************************
		No code
	********************************************************************************)
	E_ITC_SubsystemControlCode.NO_CODE:
		// No code received
		;
		
	(*******************************************************************************
		Reset error
	********************************************************************************)
	E_ITC_SubsystemControlCode.RESET_ERROR:
		// Reset Subsystem
		SubsystemData.ErrorData.Error.ResetError := TRUE;
			
	(*******************************************************************************
		Set Variable
	********************************************************************************)
	E_ITC_SubsystemControlCode.SET_VARIABLE:
		// Store variable
		ITC.Variable := SubsystemBase.SCQ.Variable;

	(*******************************************************************************
		Set Master speed request
	********************************************************************************)
	E_ITC_SubsystemControlCode.SET_MASTER_SPEED:
	
		// Check max limit master speed
		IF SubsystemBase.SCQ.Variable > SettingsSubsystem.MaxMasterSpeed THEN
			// Limit master speed
			SubsystemInterface.In.MasterSpeed := SettingsSubsystem.MaxMasterSpeed;
			
		// Check min limit master speed
		ELSIF SubsystemBase.SCQ.Variable < SettingsSubsystem.MinMasterSpeed THEN
			// Limit master speed
			SubsystemInterface.In.MasterSpeed := SettingsSubsystem.MinMasterSpeed;
		
		ELSE
			// Forward master speed
			SubsystemInterface.In.MasterSpeed := DINT_TO_INT(SubsystemBase.SCQ.Variable);
		END_IF

		F_ITC_SendSCR(
			eChannelSrc		:= meChannelSrc, 
			SubsystemName	:= F_ReduceToAlphaNumeric(SettingsSubsystem.SubsystemName), 
			Code			:= SubsystemBase.SCQ.Code, 
			Variable		:= INT_TO_DINT(SubsystemInterface.In.MasterSpeed), 
			eReturnCode		:= E_ErrorConv.NO_ERROR_CODE);

	(*******************************************************************************
		Update system time
	********************************************************************************)
	E_ITC_SubsystemControlCode.UPDATE_SYSTEM_TIME:
		// Set synchronize command
		ITC.Commands.UpdateSystemTime := TRUE;
		
		// Set time to synchronize
		SubsystemBase.TimeValue := SubsystemBase.SCQ.SystemTime;

	(*******************************************************************************
		Update all groups and positions
	********************************************************************************)
	E_ITC_SubsystemControlCode.REQUEST_GROUP_POSITION_STATUS:
		// If not already a request for a full system update is active
		IF NOT ITC.Commands.UpdateAllGroupsAndPositions THEN
			// Set command to send system update
			ITC.Commands.UpdateAllGroupsAndPositions 	:= TRUE; 
			// Store channel source
			SubsystemBase.UpdateChannelSrc := meChannelSrc;
			// Reset index
			SubsystemBase.eUpdateElementNumber := 1;
			SubsystemBase.eUpdateFunctionNumber := 1;
			SubsystemBase.eUpdateGroupNumber := 1;
		END_IF
		
ELSE
	// Unrecognised ControlRequest message received 
	DebugMsg := CONCAT('M_ITC_HandleBufferMessages - Unknown control code received: ', INT_TO_STRING(SubsystemBase.SCQ.Code));
	fbDebugMsg.M_SendErrorMsg(mMessage := DebugMsg);
END_CASE

// if request was no masterspeed cmd
IF SubsystemBase.SCQ.Code <> E_ITC_SubsystemControlCode.SET_MASTER_SPEED THEN
	F_ITC_SendSCR(
		eChannelSrc		:= meChannelSrc, 
		SubsystemName	:= F_ReduceToAlphaNumeric(SettingsSubsystem.SubsystemName), 
		Code			:= SubsystemBase.SCQ.Code, 
		Variable		:= ITC.Variable, 
		eReturnCode		:= E_ErrorConv.NO_ERROR_CODE);
END_IF
END_METHOD

METHOD PRIVATE M_ITC_SSQ : BOOL
VAR_INPUT
	meChannelSrc		: E_MFCS_CHANNEL; // Number of the source 
	mpData				: PVOID; // Data  pointer 
	mLen				: UDINT; // Data length
END_VAR
// Map data
F_BlockCopy(
	pSrc:= mpData, 
	LenSrc:= mLen, 
	pDest:= ADR(SubsystemBase.SSQ), 
	LenDest:= SIZEOF(SubsystemBase.SSQ));
	
F_ITC_SendSSR(
	eChannelSrc		:= meChannelSrc, 
	SubsystemName	:= F_ReduceToAlphaNumeric(SettingsSubsystem.SubsystemName), 
	eMode			:= SubsystemData.OperationState.eMode, 
	eState			:= SubsystemData.OperationState.eState, 
	eSystemInfo		:= E_SystemInfo.NO_INFO, 
	eErrorState		:= SubsystemData.ErrorData.ErrorState, 
	eErrorCode		:= SubsystemData.ErrorData.Error.ErrorCode.Conv, 
	eErrorType		:= SubsystemData.ErrorData.Error.ErrorType, 
	ErrorInformation:= SubsystemData.ErrorData.Error.ErrorParam, 
	Variable		:= ITC.Variable, 
	eReturnCode		:= E_ErrorConv.NO_ERROR_CODE);
END_METHOD

/// Subsystem error handler
METHOD M_MonitorSubsystemErrors : BOOL
(**************************************************************************************
 * Application   : BoxControl Framework
 * Revision date : $Date: 2020-11-19 15:59:09 +0100 (tor, 19 nov 2020) $
 * Author        : CDC
 * ------------------------------------------------------------------------------------
 * © Swisslog AG * Swisslog is not liable for any usage of this source code that is not agreed
 * on between Swisslog and the other party. The mandatory legal liability remains * unaffected.
 * ------------------------------------------------------------------------------------
 * Project revision history:
 *
 * VERSION DATE         INITIALS     DESCRIPTION
 * 0.0     DD.MM.YYYY   name       	 explain customized modifications
 *
 **************************************************************************************)
VAR
	meGroupNumber			: E_GroupNumber; // Group number
	mDataSetIdx				: INT; // Temporary data set index
	mErrorDataSet			: ST_ErrorDataSet; // Temporary error set
	mErrorData				: ST_SubsystemErrorStruct; // Temporary error data
	mGroupErrorData			: ST_GroupErrorStruct; // Group error struct
	mIdx					: INT; // Iterator
END_VAR
(**************************************************************************************************************
   Subsystem error handling
***************************************************************************************************************)

// Store current data set index
mDataSetIdx := SubsystemData.ErrorData.DataSetIdx;

// Store current error data
mErrorData := SubsystemData.ErrorData;

// Check if an error is stored
IF mDataSetIdx > 0 THEN
	// If error type has changed - Gone or changed
	IF mErrorData.ErrorDataSet[mDataSetIdx].ErrorType <> mErrorData.Error.ErrorType THEN
		
		// If the stored error type was "ERROR"
		IF mErrorData.Error.ErrorType = E_ErrorType.ERROR
           OR mErrorData.Error.ErrorType = E_ErrorType.WARNING THEN
			// Send error is gone
			ITC.Commands.NoErrorReport := TRUE;
		END_IF
		
		// Reset stored data index
		SubsystemData.ErrorData.DataSetIdx := 0;		
		
		// Reset Message
		SubsystemData.ErrorData.Error.ResetError 	:= FALSE;
		SubsystemData.ErrorData.Error.ErrorType 	:= NO_ERROR_PENDING;
		SubsystemData.ErrorData.Error.ErrorCode.Conv 	:= E_ErrorConv.NO_ERROR_CODE;
		SubsystemData.ErrorData.Error.ErrorParam 	:= '';
	END_IF
// Check if an external error is stored
ELSIF SubsystemData.ErrorData.ExternalError.ErrorType > E_ErrorType.NO_ERROR_PENDING THEN
	// If error type has changed - its gone or type has changed
	IF SubsystemData.ErrorData.ExternalError.ErrorType <> 
	   SubsystemData.ErrorData.Error.ErrorType THEN
	   
		// If the stored error type was "ERROR"
		IF SubsystemData.ErrorData.Error.ErrorType = E_ErrorType.ERROR
		   OR SubsystemData.ErrorData.Error.ErrorType = E_ErrorType.WARNING THEN
			// Send error is gone
			ITC.Commands.NoErrorReport := TRUE;
		END_IF
		
		// Reset Message
		SubsystemData.ErrorData.Error.ResetError 	:= FALSE;
		SubsystemData.ErrorData.Error.ErrorType 	:= NO_ERROR_PENDING;
		SubsystemData.ErrorData.Error.ErrorCode.Conv:= E_ErrorConv.NO_ERROR_CODE;
		SubsystemData.ErrorData.Error.ErrorParam 	:= '';
	END_IF
END_IF

(**************************************************************************************************************
   Check for new or higher prioritized message
***************************************************************************************************************)
// Loop trough all errors 
FOR mIdx := 1 TO NUMBER_OF_ERROR_SETS DO
	// Detect new or higher prioritized error message
	IF mErrorData.ErrorDataSet[mIdx].ErrorType > mErrorData.Error.ErrorType THEN
		
		// Store index of current data set
		SubsystemData.ErrorData.DataSetIdx := mIdx;
		
		// Store error data set
		mErrorDataSet := SubsystemData.ErrorData.ErrorDataSet[mIdx];
		
		// Update error
		SubsystemData.ErrorData.Error.ErrorCode.Conv := mErrorDataSet.ErrorCode.Conv;
		SubsystemData.ErrorData.Error.ErrorParam := mErrorDataSet.ErrorParam;
		SubsystemData.ErrorData.Error.ErrorType := mErrorDataSet.ErrorType;
		
		// New error - send status report
		ITC.Commands.StatusReport := TRUE;
	END_IF
	
	// Check is an error is ongoing and a reset command is set
	IF mErrorData.Error.ResetError AND 
       mErrorData.ErrorDataSet[mIdx].ErrorType <> NO_ERROR_PENDING THEN
	   
		// Reset current error data set
		SubsystemData.ErrorData.ErrorDataSet[mIdx].ResetError := TRUE;
	END_IF
END_FOR


// Check external error slot
IF SubsystemData.ErrorData.ExternalError.ErrorType > SubsystemData.ErrorData.Error.ErrorType THEN

	// Reset lower prioritized previous errors
	mDataSetIdx := 0;
	
	// Update error
	SubsystemData.ErrorData.Error.ErrorCode.Conv := SubsystemData.ErrorData.ExternalError.ErrorCode.Conv;
	SubsystemData.ErrorData.Error.ErrorParam := SubsystemData.ErrorData.ExternalError.ErrorParam;
	SubsystemData.ErrorData.Error.ErrorType := SubsystemData.ErrorData.ExternalError.ErrorType;

	// Send Report
	ITC.Commands.StatusReport := TRUE;
END_IF

// Check is an external error is ongoing and a reset command is set
IF SubsystemData.ErrorData.Error.ResetError AND 
   SubsystemData.ErrorData.ExternalError.ErrorType <> NO_ERROR_PENDING THEN

	// Reset current error data set
	SubsystemData.ErrorData.ExternalError.ResetError := TRUE;
END_IF

// If reset command is set
IF mErrorData.Error.ResetError THEN
	
	// If the stored error type was "ERROR"
	IF mErrorData.Error.ErrorType = E_ErrorType.ERROR THEN
		
		// Send error is gone
		ITC.Commands.NoErrorReport := TRUE;
	END_IF
	
	// Reset stored data index
	SubsystemData.ErrorData.DataSetIdx := 0;	

	// Reset Message
	SubsystemData.ErrorData.Error.ResetError 	:= FALSE;
	SubsystemData.ErrorData.Error.ErrorType 	:= NO_ERROR_PENDING;
	SubsystemData.ErrorData.Error.ErrorCode.Conv 	:= E_ErrorConv.NO_ERROR_CODE;
	SubsystemData.ErrorData.Error.ErrorParam 	:= '';
END_IF


(**************************************************************************************************************
   Subsystem error state
***************************************************************************************************************)

// If Subsystem is in error state
IF SubsystemData.ErrorData.Error.ErrorType = E_ErrorType.ERROR THEN
	// Set error state - ERROR
	SubsystemData.ErrorData.ErrorState := E_ErrorState.ERROR;
	
// If Subsystem is in warning state
ELSIF SubsystemData.ErrorData.Error.ErrorType = E_ErrorType.WARNING THEN
	// Set error state - WARNING
	SubsystemData.ErrorData.ErrorState := E_ErrorState.WARNING;

// If Subsystem has no error or an info is pending
ELSIF SubsystemData.ErrorData.Error.ErrorType = E_ErrorType.NO_ERROR_PENDING OR 
	  SubsystemData.ErrorData.Error.ErrorType = E_ErrorType.INFO  THEN
	// Set error state - Operational
	SubsystemData.ErrorData.ErrorState := E_ErrorState.OPERATIONAL;

ELSE
	// Otherwise -> Unknown
	SubsystemData.ErrorData.ErrorState := E_ErrorState.UNKNOWN;
END_IF

(**************************************************************************************************************
   Monitor groups
***************************************************************************************************************)
// Reset
SubsystemData.ErrorData.GroupErrorPending := FALSE;

// Go through all groups
FOR meGroupNumber := E_GroupNumber.G_BEGIN_GROUP + 1 TO E_GroupNumber.G_END_GROUP - 1 DO
	
	// Get group	
	mGroupErrorData := F_GetGroupErrorData(eGroupNumber := meGroupNumber);

	// Is group is in error state or an underlaying element
	IF mGroupErrorData.Error.ErrorType = E_ErrorType.ERROR OR
	   mGroupErrorData.ElementErrorPending THEN
	   	// Set error flag
		SubsystemData.ErrorData.GroupErrorPending := TRUE;
		EXIT;
	END_IF
END_FOR
END_METHOD

METHOD M_PreInit : BOOL
(**************************************************************************************
 * 	Application		:	BoxControl Framework
 *	Revision		:	$Revision: 404529 $
 *	Revision date	:	$Date: 2020-11-19 15:59:09 +0100 (tor, 19 nov 2020) $
 *	Last changed by	:	$Author: b7bolm $
 *	URL				:	$URL: http://almscdc.swisslog.com/repo/SWPD/Development/BoxControlFramework/20_Release/trunk/01_Software/BCF/BCF/JumpStart/20_Product/10_App/15_Subsystem/10_Lib/10_Conv/FB_SubsystemConv.TcPOU $
 *
 *	Purpose			:	Preinitialize 
 *						Clears values and load settings
 *
 * ------------------------------------------------------------------------------------
 *	Copyright Swisslog [IP AG], Switzerland. All rights reserved.
 * 
 * ------------------------------------------------------------------------------------
 *	
 * 	Revision History: 
 *
 * 	VERSION			DATE			INITIALS			DESCRIPTION
 *	0.1				01.01.2001		swl					Example
 *
 **************************************************************************************)
VAR
END_VAR
(**************************************************************************************
	Reset initialization sequence values
***************************************************************************************)
SubsystemBase.eLimitFunctionNumber := E_FunctionNumber.F_BEGIN_FUNCTION;
SubsystemBase.eLimitElementNumber := E_ElementNumber.E_BEGIN_ELEMENT;
SubsystemBase.eLimitGroupNumber := E_GroupNumber.G_BEGIN_GROUP;

(**************************************************************************************
	Load configuration
***************************************************************************************)
SettingsSubsystem := ConfigSubsystem;
END_METHOD

METHOD M_ResetError : BOOL
(**************************************************************************************
 * 	Application		:	BoxControl Framework
 *	Revision		:	$Revision: 404529 $
 *	Revision date	:	$Date: 2020-11-19 15:59:09 +0100 (tor, 19 nov 2020) $
 *	Last changed by	:	$Author: b7bolm $
 *	URL				:	$URL: http://almscdc.swisslog.com/repo/SWPD/Development/BoxControlFramework/20_Release/trunk/01_Software/BCF/BCF/JumpStart/20_Product/10_App/15_Subsystem/10_Lib/10_Conv/FB_SubsystemConv.TcPOU $
 *
 *	Purpose			:	Reset Subsystem errors.
 *
 * ------------------------------------------------------------------------------------
 *	Copyright Swisslog [IP AG], Switzerland. All rights reserved.
 * 
 * ------------------------------------------------------------------------------------
 *	
 * 	Revision History: 
 *
 * 	VERSION			DATE			INITIALS			DESCRIPTION
 *	0.1				01.01.2001		swl					Example
 *
 **************************************************************************************)
// If the Subsystem is in error
IF SubsystemData.ErrorData.Error.ErrorType  <> E_ErrorType.NO_ERROR_PENDING  THEN
	// Send reset
	SubsystemData.ErrorData.Error.ResetError := TRUE;
END_IF

M_ResetError := TRUE;
END_METHOD

METHOD M_ResetExternalError : BOOL
(**************************************************************************************
 * 	Application		:	BoxControl Framework
 *	Revision		:	$Revision: 404529 $
 *	Revision date	:	$Date: 2020-11-19 15:59:09 +0100 (tor, 19 nov 2020) $
 *	Last changed by	:	$Author: b7bolm $
 *	URL				:	$URL: http://almscdc.swisslog.com/repo/SWPD/Development/BoxControlFramework/20_Release/trunk/01_Software/BCF/BCF/JumpStart/20_Product/10_App/15_Subsystem/10_Lib/10_Conv/FB_SubsystemConv.TcPOU $
 *
 *	Purpose			:	Reset external error
 *						
 *
 * ------------------------------------------------------------------------------------
 *	Copyright Swisslog [IP AG], Switzerland. All rights reserved.
 * 
 * ------------------------------------------------------------------------------------
 *	
 * 	Revision History: 
 *
 * 	VERSION			DATE			INITIALS			DESCRIPTION
 *	0.1				01.01.2001		swl					Example
 *
 **************************************************************************************)
 VAR_INPUT
	mReset		: BOOL; // Force reset
END_VAR
// Initialize
M_ResetExternalError := FALSE;

// Reset error if ResetError command or reset command is set 
IF SubsystemData.ErrorData.ExternalError.ResetError OR mReset THEN
	// Clear error
	SubsystemData.ErrorData.ExternalError.ResetError 		:= FALSE; 
	SubsystemData.ErrorData.ExternalError.ErrorType 		:= NO_ERROR_PENDING;
	SubsystemData.ErrorData.ExternalError.ErrorCode.Conv	:= E_ErrorConv.NO_ERROR_CODE;
	SubsystemData.ErrorData.ExternalError.ErrorParam 		:= '';
	M_ResetExternalError 								:= TRUE;
END_IF
END_METHOD

METHOD M_SetExternalError : BOOL
(**************************************************************************************
 * 	Application		:	BoxControl Framework
 *	Revision		:	$Revision: 404529 $
 *	Revision date	:	$Date: 2020-11-19 15:59:09 +0100 (tor, 19 nov 2020) $
 *	Last changed by	:	$Author: b7bolm $
 *	URL				:	$URL: http://almscdc.swisslog.com/repo/SWPD/Development/BoxControlFramework/20_Release/trunk/01_Software/BCF/BCF/JumpStart/20_Product/10_App/15_Subsystem/10_Lib/10_Conv/FB_SubsystemConv.TcPOU $
 *
 *	Purpose			:	Set error
 *						Wrapped to a function to improve debugging and readability.
 *						
 *
 * ------------------------------------------------------------------------------------
 *	Copyright Swisslog [IP AG], Switzerland. All rights reserved.
 * 
 * ------------------------------------------------------------------------------------
 *	
 * 	Revision History: 
 *
 * 	VERSION			DATE			INITIALS			DESCRIPTION
 *	0.1				01.01.2001		swl					Example
 *
 **************************************************************************************)
 VAR_INPUT
	mErrorType		: E_ErrorType; // Error message type
	mErrorParam		: STRING(System.ERROR_PARAM_STRINGLENGTH); // Error parameter
	mErrorCode		: INT; // Error message
END_VAR
// Initialize
M_SetExternalError := FALSE;

// Check that the values are valid
IF mErrorType > E_ErrorType.NO_ERROR_PENDING AND mErrorCode > E_ErrorConv.NO_ERROR_CODE THEN

	SubsystemData.ErrorData.ExternalError.ErrorCode.Conv := mErrorCode;
	SubsystemData.ErrorData.ExternalError.ErrorType := mErrorType;
	SubsystemData.ErrorData.ExternalError.ErrorParam := mErrorParam;

	M_SetExternalError := TRUE;
END_IF
END_METHOD

METHOD M_UpdateRegistry
(**************************************************************************************
 * 	Application		:	BoxControl Framework
 *	Revision		:	$Revision: 404529 $
 *	Revision date	:	$Date: 2020-11-19 15:59:09 +0100 (tor, 19 nov 2020) $
 *	Last changed by	:	$Author: b7bolm $
 *	URL				:	$URL: http://almscdc.swisslog.com/repo/SWPD/Development/BoxControlFramework/20_Release/trunk/01_Software/BCF/BCF/JumpStart/20_Product/10_App/15_Subsystem/10_Lib/10_Conv/FB_SubsystemConv.TcPOU $
 *
 *	Purpose			:	Update registry information
 *
 * ------------------------------------------------------------------------------------
 *	Copyright Swisslog [IP AG], Switzerland. All rights reserved.
 * 
 * ------------------------------------------------------------------------------------
 *	
 * 	Revision History: 
 *
 * 	VERSION			DATE			INITIALS			DESCRIPTION
 *	0.1				01.01.2001		swl					Example
 *
 **************************************************************************************)
VAR_INPUT
END_VAR
VAR
	mIdx	: INT;
END_VAR

SubsystemRegistry.rSubsystemData REF= SubsystemData;
SubsystemRegistry.rSubsystemInterface REF= SubsystemInterface;
SubsystemRegistry.rSettingsSubsystem REF= SettingsSubsystem;
END_METHOD

END_FUNCTION_BLOCK

// ---- 20_Product/10_BCF/11_Conv/11_Com/11_ITC/F_ITC_SendSSR.TcPOU
FUNCTION F_ITC_SendSSR : BOOL
(**************************************************************************************
 * 	Application		:	BoxControl Framework
 *	Revision		:	$Revision: 404529 $
 *	Revision date	:	$Date: 2018-04-23 08:21:38 +0200 (Mo., 23 Apr 2018) $
 *	Last changed by	:	$Author: b7bolm $
 *	URL				:	$URL: http://almscdc.swisslog.com/repo/SWPD/Development/BoxControlFramework/20_Release/trunk/01_Software/BCF/BCF/JumpStart/20_Product/10_App/11_Com/10_Lib/10_Conv/11_ITC/F_ITC_SendSSR.TcPOU $
 *
 *	Purpose			:	Wrap message - SSR
 *
 * ------------------------------------------------------------------------------------
 *	Copyright Swisslog [IP AG], Switzerland. All rights reserved.
 * 
 * ------------------------------------------------------------------------------------
 *	
 * 	Revision History: 
 *
 * 	VERSION			DATE			INITIALS			DESCRIPTION
 *	0.1				01.01.2001		swl					Example
 *
 **************************************************************************************)
VAR_INPUT
	eChannelSrc			: E_MFCS_Channel; // Source communicaton channel	
	SubsystemName		: STRING(Conveyor.POSITION_STRINGLENGTH); // Position
	eMode				: E_PositionMode; // Mode
	eState				: E_PositionState; // State
	eSystemInfo			: E_SystemInfo; // System info
	eErrorState			: E_ErrorState; // Error State
	eErrorCode			: E_ErrorConv; // Return Code
	eErrorType			: E_ErrorType; // Error Type
	ErrorInformation	: STRING(System.ERROR_PARAM_STRINGLENGTH); // Error Information
	Variable			: DINT; // Variable
	eReturnCode			: E_ErrorConv; // Return code
END_VAR
VAR
	SSR					: ST_ITC_SSR; 
END_VAR

// Map values
SSR.SubsystemName := SubsystemName;
SSR.eMode := eMode;
SSR.eState := eState;
SSR.eSystemInfo := eSystemInfo;
SSR.eErrorState := eErrorState;
SSR.eErrorCode := eErrorCode;
SSR.eErrorType := eErrorType;
SSR.ErrorInformation := ErrorInformation;
SSR.Variable := Variable;
SSR.eReturnCode := eReturnCode;

// Forward to ITC
F_ITC_SendSSR := fbITC_Manager.M_SendData(
					meChannel	:= eChannelSrc,
					mMsgType	:= E_ITC_MsgTypeConv.SUBSYSTEM_STATUS_REPORT,
					mpData		:= ADR(SSR),
					mLen		:= SIZEOF(SSR));

END_FUNCTION

// ---- 20_Product/10_BCF/11_Conv/11_Com/11_ITC/F_ITC_SendSCR.TcPOU
FUNCTION F_ITC_SendSCR : BOOL
(**************************************************************************************
 * 	Application		:	BoxControl Framework
 *	Revision		:	$Revision: 404529 $
 *	Revision date	:	$Date: 2018-04-23 08:21:38 +0200 (Mo., 23 Apr 2018) $
 *	Last changed by	:	$Author: b7bolm $
 *	URL				:	$URL: http://almscdc.swisslog.com/repo/SWPD/Development/BoxControlFramework/20_Release/trunk/01_Software/BCF/BCF/JumpStart/20_Product/10_App/11_Com/10_Lib/10_Conv/11_ITC/F_ITC_SendSCR.TcPOU $
 *
 *	Purpose			:	Wrap message - SCR
 *
 * ------------------------------------------------------------------------------------
 *	Copyright Swisslog [IP AG], Switzerland. All rights reserved.
 * 
 * ------------------------------------------------------------------------------------
 *	
 * 	Revision History: 
 *
 * 	VERSION			DATE			INITIALS			DESCRIPTION
 *	0.1				01.01.2001		swl					Example
 *
 **************************************************************************************)
VAR_INPUT
	eChannelSrc		: E_MFCS_Channel; // Source communicaton channel		
	SubsystemName	: STRING(Conveyor.POSITION_STRINGLENGTH); // SIS Subsystem name MM-000-0000-000
	Code			: INT; // Control code
	Variable		: DINT; // Control code variable
	eReturnCode		: E_ErrorConv; // Return code
END_VAR
VAR
	SCR				: ST_ITC_SCR; 
END_VAR

// Map values
SCR.SubsystemName := SubsystemName;
SCR.Code := Code;
SCR.Variable := Variable;
SCR.ReturnCode := eReturnCode;

// Forward to ITC
F_ITC_SendSCR := fbITC_Manager.M_SendData(
					meChannel	:= eChannelSrc,
					mMsgType	:= E_ITC_MsgTypeConv.SUBSYSTEM_CONTROL_REPLY,
					mpData		:= ADR(SCR),
					mLen		:= SIZEOF(SCR));

END_FUNCTION

// ---- 20_Product/10_BCF/11_Conv/12_E_Functions/10_Helper/F_GetNumberOfZones.TcPOU
FUNCTION F_GetNumberOfZones : INT
(**************************************************************************************
 * 	Application		:	BoxControl Framework
 *	Revision		:	$Revision: 404529 $
 *	Revision date	:	$Date: 2018-04-23 08:21:38 +0200 (Mo., 23 Apr 2018) $
 *	Last changed by	:	$Author: b7bolm $
 *	URL				:	$URL: http://almscdc.swisslog.com/repo/SWPD/Development/BoxControlFramework/20_Release/trunk/01_Software/BCF/BCF/JumpStart/20_Product/10_App/12_E_Functions/10_Lib/10_Conv/10_Functions/F_GetNumberOfZones.TcPOU $
 *
 *	Purpose			:	Return number of zones
 *
 * ------------------------------------------------------------------------------------
 *	Copyright Swisslog [IP AG], Switzerland. All rights reserved.
 * 
 * ------------------------------------------------------------------------------------
 *	
 * 	Revision History: 
 *
 * 	VERSION			DATE			INITIALS			DESCRIPTION
 *	0.1				01.01.2001		swl					Example
 *
 **************************************************************************************)
VAR_INPUT
	eFunctionNumber		: E_FunctionNumber; // Function number
END_VAR

// Check if function number is valid
IF eFunctionNumber > E_FunctionNumber.F_BEGIN_FUNCTION AND
   eFunctionNumber < E_FunctionNumber.F_END_FUNCTION THEN
  
   // Check reference is valid
   IF __ISVALIDREF(FunctionRegistry[eFunctionNumber].rSettingsFunction) THEN
		// Return number
		F_GetNumberOfZones := FunctionRegistry[eFunctionNumber].rSettingsFunction.NumberOfZones;
   END_IF
END_IF

END_FUNCTION

// ---- 20_Product/10_BCF/11_Conv/14_Groups/10_Helper/F_GetGroupErrorData.TcPOU
FUNCTION F_GetGroupErrorData : ST_GroupErrorStruct
(**************************************************************************************
 * 	Application		:	BoxControl Framework
 *	Revision		:	$Revision: 404529 $
 *	Revision date	:	$Date: 2018-04-23 08:21:38 +0200 (Mo., 23 Apr 2018) $
 *	Last changed by	:	$Author: b7bolm $
 *	URL				:	$URL: http://almscdc.swisslog.com/repo/SWPD/Development/BoxControlFramework/20_Release/trunk/01_Software/BCF/BCF/JumpStart/20_Product/10_App/14_Groups/10_Lib/10_Conv/10_Functions/F_GetGroupErrorData.TcPOU $
 *
 *	Purpose			:	Return group error data
 *
 * ------------------------------------------------------------------------------------
 *	Copyright Swisslog [IP AG], Switzerland. All rights reserved.
 * 
 * ------------------------------------------------------------------------------------
 *	
 * 	Revision History: 
 *
 * 	VERSION			DATE			INITIALS			DESCRIPTION
 *	0.1				01.01.2001		swl					Example
 *
 **************************************************************************************)
VAR_INPUT
	eGroupNumber		: E_GroupNumber; // Group number
END_VAR


// Check if group number is valid
IF eGroupNumber > E_GroupNumber.G_BEGIN_GROUP AND
   eGroupNumber < E_GroupNumber.G_END_GROUP THEN

	// Check reference is valid
	IF __ISVALIDREF(GroupRegistry[eGroupNumber].rGroup) THEN
   		// Return error data
   		F_GetGroupErrorData := GroupRegistry[eGroupNumber].rGroup.GroupData.ErrorData;
	END_IF
END_IF

END_FUNCTION

// ---- 20_Product/30_Toolbox/99_Misc/FB_SystemInfo.TcPOU
FUNCTION_BLOCK FB_SystemInfo
(**************************************************************************************
 * 	Application		:	BoxControl Framework
 *	Revision		:	$Revision: 404529 $
 *	Revision date	:	$Date: 2018-04-23 08:21:38 +0200 (Mo., 23 Apr 2018) $
 *	Last changed by	:	$Author: b7bolm $
 *	URL				:	$URL: http://almscdc.swisslog.com/repo/SWPD/Development/BoxControlFramework/20_Release/trunk/01_Software/BCF/BCF/JumpStart/30_Toolbox/99_Misc/FB_SystemInfo.TcPOU $
 *
 *	Purpose			:	This functionblock should provide information about the system.
 *
 * ------------------------------------------------------------------------------------
 *	Copyright Swisslog [IP AG], Switzerland. All rights reserved.
 * 
 * ------------------------------------------------------------------------------------
 *	
 * 	Revision History: 
 *
 * 	VERSION			DATE			INITIALS			DESCRIPTION
 *	0.1				01.01.2001		swl					Example
 *
 **************************************************************************************)
VAR_INPUT
	TimeInterval 		: TIME := T#5S; // Polling time
END_VAR
VAR_OUTPUT
	Error				: BOOL; // Error during data gathering
	CPU_Temperatur		: INT; // Current cpu temperatur
	CPU_Usage			: INT; // Current cpu usage
	SystemUsage			: INT; // Current system usage
	FanSpeed			: UINT; // Fan speed
END_VAR
VAR
	fbTimeIntervalCPU	: TON; // Interval for gathering CPU data
	fbTimeIntervalSystem: TON; // Interval for gathering system data
	eCpuStates			: E_CPU_InfoStates;
	fbGetCPU 			: FB_MDP_CPU_Read;
	fbGetCpuTemp		: FB_MDP_ReadElement;
	fbGetCpuUsage		: FB_MDP_ReadElement;
	fbGetFanSpeed		: FB_MDP_ReadElement;
	CPU_MDP_Addr		: ST_MDP_Addr;
	HeaderCPU_Mod		: ST_MDP_ModuleHeader;
	ContentCPU_Mod		: ST_MDP_CPU;
	fbSystemLatency		: TC_SysLatency;
END_VAR


(**************************************************************************************************************
   Gathering CPU data
***************************************************************************************************************)
A_CPU();

(**************************************************************************************************************
   Gathering System data
***************************************************************************************************************)
A_System();

ACTION A_CPU:
(**************************************************************************************
 * 	NAME		A_CPU
 * 	FUNCTION	Gathering data of CPU
 **************************************************************************************)
 
CASE eCpuStates OF
	
	(**************************************************************************************
   		Init
	***************************************************************************************)
	E_CPU_InfoStates.INIT:
		fbTimeIntervalCPU(IN := FALSE);

		// Change state
		eCpuStates := E_CPU_InfoStates.READ_DEVICE;
			
	(**************************************************************************************
   		Read device (CPU)
	***************************************************************************************)
	E_CPU_InfoStates.READ_DEVICE:
	
		fbTimeIntervalCPU(IN := TRUE, PT := TimeInterval);
		
		IF fbTimeIntervalCPU.Q THEN
			// Reset
			Error := FALSE;
			
			// Get access to CPU 0
			fbGetCPU(
				bExecute	:= TRUE,
				iModIdx   	:= 0,	
				sAmsNetId 	:= '');
				
			// Change state
			eCpuStates := E_CPU_InfoStates.READ_TEMPERATURE;
		END_IF
	
	(**************************************************************************************
   		Read temperature
	***************************************************************************************)
	E_CPU_InfoStates.READ_TEMPERATURE:
		fbGetCPU(bExecute	:= FALSE);
		
		// Wait until fbGetCPU is done
		IF NOT fbGetCPU.bBusy THEN
			// Error occured
			IF fbGetCPU.bError THEN
				// Set error
				Error := TRUE;
				
				// Change state
				eCpuStates := E_CPU_InfoStates.INIT;
			ELSE
				// Store address info
				HeaderCPU_Mod := fbGetCPU.stMDP_ModuleHeader;
				ContentCPU_Mod := fbGetCPU.stMDP_ModuleContent;
				
				// Define element of CPU temperature
				CPU_MDP_Addr.nArea := INT_TO_BYTE(eMDP_Area_ConfigArea);
				CPU_MDP_Addr.nTableId := 1;
				CPU_MDP_Addr.nSubIdx := 3; // Temperatur
				
				// Read CPU Temperatur
				fbGetCpuTemp(
					bExecute 	:= TRUE,
					eModuleType := E_MDP_ModuleType.eMDP_ModT_CPU,
					stMDP_Addr  := CPU_MDP_Addr,
					iModIdx     := 0,
					pDstBuf     := ADR(CPU_Temperatur),
					cbDstBufLen := SIZEOF(CPU_Temperatur),
					sAmsNetId   := '');
			
				// Change state
				eCpuStates := E_CPU_InfoStates.READ_USAGE;
			END_IF
		END_IF
	
	(**************************************************************************************
   		Read latency
	***************************************************************************************)
	E_CPU_InfoStates.READ_USAGE:
		fbGetCpuTemp(bExecute := FALSE);
		
		// Wait until fbGetCpuTemp is done
		IF NOT fbGetCpuTemp.bBusy THEN
			// Error occured
			IF fbGetCpuTemp.bError THEN
				// Set error
				Error := TRUE;
				
				// Change state
				eCpuStates := E_CPU_InfoStates.INIT;
			ELSE
				// Define element of CPU temperature
				CPU_MDP_Addr.nArea := INT_TO_BYTE(eMDP_Area_ConfigArea);
				CPU_MDP_Addr.nTableId := 1;
				CPU_MDP_Addr.nSubIdx := 2; // Usage
				
				// Read CPU Usage
				fbGetCpuUsage(
					bExecute    := TRUE,
					eModuleType := E_MDP_ModuleType.eMDP_ModT_CPU,	
					stMDP_Addr  := CPU_MDP_Addr,
					iModIdx     := 0,
					pDstBuf     := ADR(CPU_Usage),
					cbDstBufLen := SIZEOF(CPU_Usage),
					sAmsNetId   := '');
					
				// Change state
				eCpuStates := E_CPU_InfoStates.READ_FAN;
			END_IF
		END_IF
	(**************************************************************************************
   		Read FAN speed
	***************************************************************************************)
	E_CPU_InfoStates.READ_FAN:
		fbGetCpuUsage(bExecute := FALSE);
		
		// Wait until fbGetCpuUsage is done
		IF NOT fbGetCpuUsage.bBusy THEN
			// Set error
			IF fbGetCpuUsage.bError THEN
				Error := TRUE;
				
				// Change state
				eCpuStates := E_CPU_InfoStates.INIT;
			ELSE
				// Define element of CPU temperature
				CPU_MDP_Addr.nArea := INT_TO_BYTE(eMDP_Area_ConfigArea);
				CPU_MDP_Addr.nTableId := 1;
				CPU_MDP_Addr.nSubIdx := 1; // Fan
				
				// Read FAN speed
				fbGetFanSpeed(
					bExecute    := TRUE,
					eModuleType := E_MDP_ModuleType.eMDP_ModT_Fan,	
					stMDP_Addr  := CPU_MDP_Addr,
					iModIdx     := 0,
					pDstBuf     := ADR(FanSpeed),
					cbDstBufLen := SIZEOF(FanSpeed),
					sAmsNetId   := '');	
			END_IF
			
			// Change state
			eCpuStates := E_CPU_InfoStates.DONE;
		END_IF
		
	(**************************************************************************************
   		Done
	***************************************************************************************)
	E_CPU_InfoStates.DONE:
		fbGetFanSpeed(bExecute := FALSE);
		
		// Wait until fbGetCpuUsage is done
		IF NOT fbGetFanSpeed.bBusy THEN
			// Set error
			Error := fbGetCpuUsage.bError;
			
			// Change state
			eCpuStates := E_CPU_InfoStates.INIT;
		END_IF
	
ELSE
	// Default go to INIT
	eCpuStates := E_CPU_InfoStates.INIT;
END_CASE
END_ACTION

ACTION A_System:
(**************************************************************************************
 * 	NAME		A_System
 * 	FUNCTION	Gathering data of CPU
 **************************************************************************************)
 
fbTimeIntervalSystem(IN := NOT fbSystemLatency.BUSY, PT := TimeInterval);

 // Get System Latency
fbSystemLatency(Start := fbTimeIntervalSystem.Q AND NOT fbSystemLatency.BUSY);
END_ACTION

END_FUNCTION_BLOCK

// ---- 20_Product/10_BCF/11_Conv/10_Base/F_MonitorEtherCAT_Master.TcPOU
FUNCTION F_MonitorEtherCAT_Master : BOOL
(**************************************************************************************
 * 	Application		:	BoxControl Framework
 *	Revision		:	$Revision: 404529 $
 *	Revision date	:	$Date: 2018-04-23 08:21:38 +0200 (Mo., 23 Apr 2018) $
 *	Last changed by	:	$Author: b7bolm $
 *	URL				:	$URL: http://almscdc.swisslog.com/repo/SWPD/Development/BoxControlFramework/20_Release/trunk/01_Software/BCF/BCF/JumpStart/20_Product/10_App/10_Base/10_Lib/10_Conv/F_MonitorEtherCAT_Master.TcPOU $
 *
 *	Purpose			:	Reads the actual EtherCAT state of the element node and decodes 
 *						node communication state and error state
 *
 * ------------------------------------------------------------------------------------
 *	Copyright Swisslog [IP AG], Switzerland. All rights reserved.
 * 
 * ------------------------------------------------------------------------------------
 *	
 * 	Revision History: 
 *
 * 	VERSION			DATE			INITIALS			DESCRIPTION
 *	0.1				01.01.2001		swl					Example
 *
 **************************************************************************************)
VAR_INPUT
	MasterDeviceState			: E_EtherCAT_MasterError; // Device state
	MasterDeviceWorkingCounter	: UINT; // Working counter (Telegram lost)
END_VAR

VAR_IN_OUT
	ErrorData					: ST_ErrorDataSet; // Error data 
END_VAR

(*
0x0001 = Link error
0x0002 = I/O locked after link error (I/O reset required)
0x0004 = Link error (redundancy adapter)
0x0008 = Missing one frame (redundancy mode)
0x0010 = Out of send resources (I/O reset required)
0x0020 = Watchdog triggered
0x0040 = Ethernet driver (miniport) not found
0x0080 = I/O reset active
0x0100 = At least one device in 'INIT' state
0x0200 = At least one device in 'PRE-OP' state
0x0400 = At least one device in 'SAFE-OP' state
0x0800 = At least one device indicates an error state
0x1000 = DC not in sync
*)

// Reset error  
F_ResetError(Reset := FALSE, ErrorData := ErrorData);

// Set error 
IF MasterDeviceState <> ETHERCAT_MASTER_NO_ERROR THEN
	ErrorData.ErrorCode.Conv:= E_ErrorConv.ETHERCAT_MASTER_ERROR;
	ErrorData.ErrorType 	:= E_ErrorType.ERROR;
	ErrorData.ErrorParam 	:= INT_TO_STRING(MasterDeviceState);
END_IF

// Working counter
IF MasterDeviceWorkingCounter > 0 THEN
	ErrorData.ErrorCode.Conv:= E_ErrorConv.ETHERCAT_MASTER_TELEGRAM_LOST;
	ErrorData.ErrorType 	:= E_ErrorType.WARNING;
	ErrorData.ErrorParam 	:= UINT_TO_STRING(MasterDeviceWorkingCounter);
END_IF

END_FUNCTION

// ---- 10_Project/10_App/12_FlowControl/FB_MergingService.TcPOU
FUNCTION_BLOCK FB_MergingService
VAR_INPUT
	///Calling function number
	eFunctionNumber: E_FunctionNumber;
END_VAR
VAR
	///Debug message service
	fbDebugMsg: FB_DebugMsg;
	///Debug message
	DebugMsg: T_MAXSTRING;
	///Merging service routines for group 1
	fbMergingService_001: FB_MergingService_001;
END_VAR
VAR_OUTPUT
	///Result previous function number
	ePrevFunctionNumber: E_FunctionNumber;
END_VAR


// Example 
// Initialize variable
ePrevFunctionNumber := F_BEGIN_FUNCTION;

CASE eFunctionNumber OF
	
	E_FunctionNumber.F_10_001_0200_01_0 .. E_FunctionNumber.F_10_001_0233_01_0:
		fbMergingService_001(
			eFunctionNumber := eFunctionNumber,
			ePrevFunctionNumber => ePrevFunctionNumber);
			
//	E_FunctionNumber.F_10_002_1250_01_0 .. E_FunctionNumber.F_10_002_1250_02_0:
//		fbMergingService_002(
//			eFunctionNumber := eFunctionNumber,
//			ePrevFunctionNumber => ePrevFunctionNumber);
	
ELSE
	DebugMsg := CONCAT('Merging area not defined. FunctionNumber: ', INT_TO_STRING(eFunctionNumber));
	fbDebugMsg.M_SendInfoMsg(DebugMsg);
END_CASE

END_FUNCTION_BLOCK

// ---- 10_Project/10_App/12_FlowControl/FB_MergingService_001.TcPOU
FUNCTION_BLOCK FB_MergingService_001
VAR_INPUT
	///Calling function number
	eFunctionNumber: E_FunctionNumber;
END_VAR
VAR
	///Debug message service
	fbDebugMsg: FB_DebugMsg;
	///Debug message
	DebugMsg: T_MAXSTRING;
	FlipFlopBool : BOOL;
	PrevZone : ST_ZoneData;
END_VAR
VAR_OUTPUT
	///Result previous function number
	ePrevFunctionNumber: E_FunctionNumber;
END_VAR


// Example 
// Initialize variable
ePrevFunctionNumber := F_BEGIN_FUNCTION;

CASE eFunctionNumber OF
	
	E_FunctionNumber.F_10_001_0200_01_0:
		IF(F_PB_GetTuDestination(eFunctionNumber:= F_10_001_0201_01_0, 1,1) = E_FunctionNumber.F_10_001_0200_01_0) THEN
			ePrevFunctionNumber := F_10_001_0201_01_0;
		END_IF
		
	E_FunctionNumber.F_10_001_0209_01_0:
		PrevZone := F_GetZoneData(E_FunctionNumber.F_10_001_0208_01_0, 1);
		IF PrevZone.TransportControlData.Occupied THEN
			ePrevFunctionNumber := F_10_001_0208_01_0;
		ELSE 
			ePrevFunctionNumber := F_10_001_0227_01_0;
		END_IF
		
	E_FunctionNumber.F_10_001_0212_01_0:
		PrevZone := F_GetZoneData(E_FunctionNumber.F_10_001_0211_01_0, 1);
		IF PrevZone.TransportControlData.Occupied THEN
			ePrevFunctionNumber := F_10_001_0211_01_0;
		ELSE 
			ePrevFunctionNumber := F_10_001_0217_01_0;
		END_IF
	

//	E_FunctionNumber.F_10_001_0221_01_0:
//		PrevZone := F_GetZoneData(E_FunctionNumber.F_10_001_0211_01_0, 1);
//		IF PrevZone.TransportControlData.Occupied THEN
//			ePrevFunctionNumber := F_10_001_0211_01_0;
//		ELSE 
//			ePrevFunctionNumber := F_10_001_0217_01_0;
//		END_IF

ELSE
	DebugMsg := CONCAT('Merging function not defined. FunctionNumber: ', INT_TO_STRING(eFunctionNumber));
	fbDebugMsg.M_SendInfoMsg(DebugMsg);
END_CASE

END_FUNCTION_BLOCK

// ---- 20_Product/20_ProBox/30_Toolbox/F_PB_GetTuDestination.TcPOU
FUNCTION F_PB_GetTuDestination : E_FunctionNumber
VAR_INPUT
	eFunctionNumber		: E_FunctionNumber; // Function number
	ZoneNumber			: INT; // ZoneNumber
	TuTableDestIdx		: INT; // Which Tu Table destination slot (Default 1)
END_VAR
VAR_OUTPUT	
	TU_DataIndex		: DINT;
END_VAR


IF( ZoneNumber > 0 AND ZoneNumber <= Conveyor.NUMBER_OF_ZONES_PER_FUNCTION) THEN

		// If zone is valid and consists of a TU-Data index
		IF __ISVALIDREF(FunctionRegistry[eFunctionNumber].Zone[ZoneNumber].refZoneData) THEN
			TU_DataIndex := FunctionRegistry[eFunctionNumber].Zone[ZoneNumber].refZoneData.TransportControlData.TU_DataIndex;
			 IF TU_DataIndex > 0 THEN
				// Return destination slot
				F_PB_GetTuDestination := TU_DataTable[TU_DataIndex].Destination[TuTableDestIdx].eFunctionNumber;				
			 END_IF
		END_IF	
END_IF

END_FUNCTION

// ---- 20_Product/10_BCF/11_Conv/12_E_Functions/10_Helper/F_GetZoneData.TcPOU
FUNCTION F_GetZoneData : ST_ZoneData
(**************************************************************************************
 * 	Application		:	BoxControl Framework
 *	Revision		:	$Revision: 404529 $
 *	Revision date	:	$Date: 2018-04-23 08:21:38 +0200 (Mo., 23 Apr 2018) $
 *	Last changed by	:	$Author: b7bolm $
 *	URL				:	$URL: http://almscdc.swisslog.com/repo/SWPD/Development/BoxControlFramework/20_Release/trunk/01_Software/BCF/BCF/JumpStart/20_Product/10_App/12_E_Functions/10_Lib/10_Conv/10_Functions/F_GetZoneData.TcPOU $
 *
 *	Purpose			:	Return zone data
 *
 * ------------------------------------------------------------------------------------
 *	Copyright Swisslog [IP AG], Switzerland. All rights reserved.
 * 
 * ------------------------------------------------------------------------------------
 *	
 * 	Revision History: 
 *
 * 	VERSION			DATE			INITIALS			DESCRIPTION
 *	0.1				01.01.2001		swl					Example
 *
 **************************************************************************************)
VAR_INPUT
	eFunctionNumber		: E_FunctionNumber;
	ZoneNumber			: INT; 
END_VAR
VAR
	ZoneData			: ARRAY[1..NUMBER_OF_ZONES_PER_FUNCTION] OF ST_ZoneData; // all zone data
END_VAR



// Check if function number and zone is valid
IF eFunctionNumber > E_FunctionNumber.F_BEGIN_FUNCTION AND
   eFunctionNumber < E_FunctionNumber.F_END_FUNCTION AND
   ZoneNumber > 0 AND ZoneNumber <= NUMBER_OF_ZONES_PER_FUNCTION THEN
  
	// Check reference is valid
    IF __ISVALIDREF(FunctionRegistry[eFunctionNumber].rFunction) THEN
	   // Return zone data
	   F_GetZoneData := FunctionRegistry[eFunctionNumber].rFunction.ZoneData[ZoneNumber];
    END_IF  
END_IF

END_FUNCTION

// ---- 10_Project/10_App/12_FlowControl/FB_RoutingService.TcPOU
FUNCTION_BLOCK FB_RoutingService
VAR_INPUT
	///Calling function number
	eFunctionNumber: E_FunctionNumber;
END_VAR
VAR
	///Debug message service
	fbDebugMsg: FB_DebugMsg;
	///Debug message
	DebugMsg: T_MAXSTRING;
	///Routing service routines for group 1
	fbRoutingService_001: FB_RoutingService_001;
END_VAR
VAR_OUTPUT
	///Result next function number
	eNextFunctionNumber: E_FunctionNumber;
END_VAR


// Example 
// Initialize variable
eNextFunctionNumber := F_BEGIN_FUNCTION;

CASE eFunctionNumber OF
	
	E_FunctionNumber.F_10_001_0200_01_0 .. E_FunctionNumber.F_10_001_0233_01_0:
		fbRoutingService_001(
			eFunctionNumber := eFunctionNumber,
			eNextFunctionNumber => eNextFunctionNumber);	

//	E_FunctionNumber.F_10_002_1250_01_0 .. E_FunctionNumber.F_10_002_1250_02_0:
//		fbRoutingService_002(
//			eFunctionNumber := eFunctionNumber,
//			eNextFunctionNumber => eNextFunctionNumber);		

ELSE
	DebugMsg := CONCAT('Routing area not defined. FunctionNumber: ', INT_TO_STRING(eFunctionNumber));
	fbDebugMsg.M_SendInfoMsg(DebugMsg);
END_CASE

END_FUNCTION_BLOCK

// ---- 10_Project/10_App/12_FlowControl/FB_RoutingService_001.TcPOU
FUNCTION_BLOCK FB_RoutingService_001
VAR_INPUT
	///Calling function number
	eFunctionNumber: E_FunctionNumber;
END_VAR
VAR
	///Debug message service
	fbDebugMsg: FB_DebugMsg;
	///Debug message
	DebugMsg: T_MAXSTRING;
	NextZone : ST_ZoneData;
	TUDest : E_FunctionNumber;
END_VAR
VAR_OUTPUT
	///Result next function number
	eNextFunctionNumber: E_FunctionNumber;
END_VAR


// Example 
// Initialize variable
eNextFunctionNumber := F_BEGIN_FUNCTION;

CASE eFunctionNumber OF
	
	E_FunctionNumber.F_10_001_0200_01_0:
		IF(F_PB_GetTuDestination(eFunctionNumber:= eFunctionNumber, 1,1) = E_FunctionNumber.F_10_001_0203_01_0) THEN
			eNextFunctionNumber := E_FunctionNumber.F_10_001_0201_01_0;
		END_IF
		
	E_FunctionNumber.F_10_001_0203_01_0:
		NextZone := F_GetZoneData(E_FunctionNumber.F_10_001_0204_01_0, 1);
		IF NOT NextZone.TransportControlData.Occupied THEN
			eNextFunctionNumber := E_FunctionNumber.F_10_001_0204_01_0;
		END_IF
	
	E_FunctionNumber.F_10_001_0204_01_0:
		IF(F_PB_GetTuDestination(eFunctionNumber:= eFunctionNumber, 1,1) = E_FunctionNumber.F_10_001_0233_01_0) THEN
			eNextFunctionNumber := E_FunctionNumber.F_10_001_0233_01_0;
		ELSE
			eNextFunctionNumber := E_FunctionNumber.F_10_002_0206_01_0;
		END_IF
		
	E_FunctionNumber.F_10_001_0209_01_0:
		IF(F_PB_GetTuDestination(eFunctionNumber:= eFunctionNumber, 1,1) = E_FunctionNumber.F_10_001_0215_02_0) THEN
			eNextFunctionNumber := E_FunctionNumber.F_10_001_0214_01_0;
		ELSE
			eNextFunctionNumber := E_FunctionNumber.F_10_001_0211_01_0;
		END_IF
		
	E_FunctionNumber.F_10_001_0212_01_0:
		IF(F_PB_GetTuDestination(eFunctionNumber:= eFunctionNumber, 1,1) = E_FunctionNumber.F_10_001_0213_01_0) THEN
			eNextFunctionNumber := E_FunctionNumber.F_10_001_0213_01_0;
		ELSE
			eNextFunctionNumber := E_FunctionNumber.F_10_001_0218_01_0;
		END_IF
		
	E_FunctionNumber.F_10_001_0222_01_0:
		TUDest := F_PB_GetTuDestination(eFunctionNumber:= eFunctionNumber, 1,1);
		IF TUDest = E_FunctionNumber.F_10_001_0232_01_0 OR TUDest = E_FunctionNumber.F_10_001_0207_01_0 THEN
			eNextFunctionNumber := E_FunctionNumber.F_10_001_0230_01_0;
		ELSE
			eNextFunctionNumber := E_FunctionNumber.F_10_001_0225_01_0;
		END_IF
ELSE
	DebugMsg := CONCAT('Routing function not defined. FunctionNumber: ', INT_TO_STRING(eFunctionNumber));
	fbDebugMsg.M_SendInfoMsg(DebugMsg);
END_CASE

END_FUNCTION_BLOCK

// ---- 20_Product/20_ProBox/22_ProMove/14_Groups/11_Emu/FB_ProBOXSG_Emulation.TcPOU
FUNCTION_BLOCK FB_ProBOXSG_Emulation EXTENDS FB_GroupConvEmulation
(**************************************************************************************
 * 	Application		:	BoxControl Framework
 *	Revision		:	$Revision: 417092 $
 *	Revision date	:	$Date: 2018-11-14 12:58:58 +0100 (Mi., 14 Nov 2018) $
 *	Last changed by	:	$Author: q8aberh $
 *	URL				:	$URL: http://almscdc.swisslog.com/repo/SWPD/Development/ProMove/02_Controls/ProBox/03_Implementation/01_DevelopmentProject/01_Software/ProBox_COE/ProBox_DevProj_v1.0/PLC_1/20_Product/11_Emu/14_Groups/10_Lib/10_Conv/FB_DummySG_Emulation.TcPOU $
 *
 *	Purpose			:	Emulation switching group.
 *
 * ------------------------------------------------------------------------------------
 *	Copyright Swisslog [IP AG], Switzerland. All rights reserved.
 * 
 * ------------------------------------------------------------------------------------
 *	
 * 	Revision History: 
 *
 * 	VERSION			DATE			INITIALS			DESCRIPTION
 *	0.1				01.01.2001		swl					Example
 *
 **************************************************************************************)
VAR_INPUT
	Config						: ST_CFG_ProBoxSGEmulation; // Configuration emulation
END_VAR
 
VAR
	pGroup						: POINTER TO FB_ProBOXSG; // Address to Group
	rGroup						: REFERENCE TO FB_ProBOXSG; // Reference to real instance
	DebugResetButton			: BOOL; //for debug purpose or visualisation
	DebugStartButton			: BOOL; //for debug purpose or visualisation
	DebugManualModeSw			: BOOL; //for debug purpose or visualisation
	DebugResetEmgButton			: BOOL; //for debug purpose or visualisation
	DebugMcOnButton				: BOOL; //for debug purpose or visualisation
	
	EmgStatus 					: ST_EmgStatus :=(eInternal:=TRUE, eExternal:=TRUE, eInternError:=FALSE);
END_VAR

VAR PERSISTENT
	Settings					: ST_CFG_ProBoxSGEmulation; // Settings 
END_VAR


(**************************************************************************************************************
   Initialization
***************************************************************************************************************)
A_Init();


(**************************************************************************************************************
   Update reference
***************************************************************************************************************)
A_UpdateReference();


(**************************************************************************************************************
   Emulation
***************************************************************************************************************)
// If emulation group is initialized
IF GroupData.Init THEN
	
	// Update real data
	M_UpdateRealObjectData();	

	// Overwrite inputs
	A_OverWriteInputs();
END_IF

ACTION A_Init:
(**************************************************************************************
 * 	NAME		A_Init
 * 	FUNCTION	Initialize emulated group
 **************************************************************************************)
 
// If group is not initialized
IF NOT GroupData.Init THEN

	// Check that linked group number is valid
	IF eGroupNumber > E_GroupNumber.G_BEGIN_GROUP AND
	   eGroupNumber < E_GroupNumber.G_END_GROUP THEN

		// Load emulation settings	
		Settings := Config;
		
		// Check that the real module is initialized
		IF F_IsGroupInitialized(eGroupNumber := eGroupNumber) THEN
			// Module is initialized
			GroupData.Init := TRUE;
			
			// Send debug message
			DebugMsg := CONCAT('Initialization done. Group: ', GroupRegistry[eGroupNumber].GroupName);
			fbDebugMsg.M_SendInfoMsg(DebugMsg);
			
			// Initialize real module
			F_InitializeGroup(eGroupNumber := eGroupNumber);
		END_IF
	END_IF
END_IF
END_ACTION

ACTION A_OverWriteInputs:
(**************************************************************************************
 * 	NAME		A_OverWriteInputs
 * 	FUNCTION	Overwrite inputs for emulation
 **************************************************************************************)

 // Modes
rGroup.HW_Inputs.AK.OpManAuto				:= NOT DebugManualModeSw;

// Commands
rGroup.HW_Inputs.AK.OpResetError			:= DebugResetButton;
rGroup.HW_Inputs.AK.OpAutoOn				:= (Settings.Autostart AND NOT GroupRegistry[rGroup.ConfigGroup.eGroupNumber].rGroupData.Init) OR DebugStartButton;
rGroup.HW_Inputs.AK.OpMcOff					:= TRUE; //NC Push button
//rGroup.HW_Inputs.AK.Ext.OpEntryReq				:= TRUE; //NC Auto/EntryRequest.

// Device input states
MemSet(ADR(rGroup.HW_Inputs.Diag.FeedBackMainContactorOFF),0,SIZEOF(rGroup.HW_Inputs.Diag.FeedBackMainContactorOFF));

rGroup.HW_Inputs.Diag.FireAlarm						:= TRUE;
rGroup.HW_Inputs.Diag.SupplyCircuitBreaker			:= TRUE;
rGroup.HW_Inputs.Diag.ASI_BusConfigError				:= FALSE;

DebugResetButton:=FALSE;

//Set Emergency status to "ok"
rGroup.M_SetEmgStatus(EmgStatus);//EmergencyCircuitOK
END_ACTION

ACTION A_UpdateReference:
(**************************************************************************************
 * 	NAME		A_UpdateReference
 * 	FUNCTION	Update reference to real object
 **************************************************************************************)

// Check valid group number
IF eGroupNumber > E_GroupNumber.G_BEGIN_GROUP AND
   eGroupNumber < E_GroupNumber.G_END_GROUP THEN

	// Is reference valid  
	IF __ISVALIDREF(GroupRegistry[eGroupNumber].rGroup) THEN
		// Build address to reference
		pGroup := ADR(GroupRegistry[eGroupNumber].rGroup);

		// If address is possible
		IF pGroup <> 0 THEN
			// Build reference to memory
			rGroup REF= pGroup^;
		ELSE
			// Reinitialize module
			GroupData.Init := FALSE;
		END_IF
	ELSE
		// Reinitialize module
		GroupData.Init := FALSE;
	END_IF
END_IF
END_ACTION

END_FUNCTION_BLOCK

// ---- 20_Product/10_BCF/11_Conv/14_Groups/09_Emulation/FB_GroupConvEmulation.TcPOU
FUNCTION_BLOCK FB_GroupConvEmulation EXTENDS FB_BaseObjectEmulation
(**************************************************************************************
 * 	Application		:	BoxControl Framework
 *	Revision		:	$Revision: 404529 $
 *	Revision date	:	$Date: 2018-04-23 08:21:38 +0200 (Mo., 23 Apr 2018) $
 *	Last changed by	:	$Author: b7bolm $
 *	URL				:	$URL: http://almscdc.swisslog.com/repo/SWPD/Development/BoxControlFramework/20_Release/trunk/01_Software/BCF/BCF/JumpStart/20_Product/11_Emu/14_Groups/10_Lib/10_Conv/FB_GroupConvEmulation.TcPOU $
 *
 *	Purpose			:	Base Group - Emulation.
 *
 * ------------------------------------------------------------------------------------
 *	Copyright Swisslog [IP AG], Switzerland. All rights reserved.
 * 
 * ------------------------------------------------------------------------------------
 *	
 * 	Revision History: 
 *
 * 	VERSION			DATE			INITIALS			DESCRIPTION
 *	0.1				01.01.2001		swl					Example
 *
 **************************************************************************************)
VAR_INPUT
	eGroupNumber				: E_GroupNumber; // Group enum link
END_VAR

VAR
	GroupBase					: ST_GroupBaseEmulation;
END_VAR

VAR PERSISTENT
	GroupData					: ST_GroupDataEmulation; // Element data emulation
END_VAR

(**************************************************************************************************************
   Group Emulation - Body never called!
***************************************************************************************************************)
;

METHOD PRIVATE M_ITC_ERQ : BOOL
VAR_INPUT
	meChannelSrc		: E_MFCS_CHANNEL; // Number of the source 
	mpData				: PVOID; // Data  pointer 
	mLen				: UDINT; // Data length
END_VAR
// Map data
F_BlockCopy(
	pSrc:= mpData, 
	LenSrc:= mLen, 
	pDest:= ADR(GroupBase.ERQ), 
	LenDest:= SIZEOF(GroupBase.ERQ));		

// Send "Error" request
GroupData.ITC.Commands.Error :=  GroupBase.ERQ.Code = 0;
GroupData.ITC.Commands.ErrorCode := GroupBase.ERQ.ErrorCode;
END_METHOD

METHOD M_ITC_ProcessMsg : BOOL
VAR_INPUT
	meChannelSrc		: E_MFCS_CHANNEL; // Number of the source 
	mMsgType			: INT; // Message type
	mpData				: PVOID; // Data  pointer 
	mLen				: UDINT; // Data length
END_VAR

// Initialize
M_ITC_ProcessMsg := TRUE;

// Validate inputs
IF mpData > 0 AND
   mLen > 0 THEN
	// map enum
	GroupBase.eMsgType := mMsgType;

	// Validate message type
	CASE GroupBase.eMsgType OF

		(*******************************************************************************
		  No Message
		********************************************************************************)
		E_ITC_MsgTypeConv.NO_MESSAGE_TYPE:
			// Empty message received
			DebugMsg := 'Empty ITC message received.';
			fbDebugMsg.M_SendErrorMsg(DebugMsg);
			
		(*******************************************************************************
		  Modify error 
		********************************************************************************)
		E_ITC_MsgTypeConv.E_ERROR_REQUEST:
			M_ITC_ERQ(meChannelSrc := meChannelSrc, mpData := mpData, mLen := mLen);

	ELSE
		// Unknown ITC message type received
		DebugMsg := CONCAT('Group emulation unknown ITC Message type: ', INT_TO_STRING(GroupBase.eMsgType));
		fbDebugMsg.M_SendErrorMsg(DebugMsg);
	END_CASE
END_IF
END_METHOD

METHOD M_UpdateRealObjectData
(**************************************************************************************
 * 	Application		:	BoxControl Framework
 *	Revision		:	$Revision: 404529 $
 *	Revision date	:	$Date: 2018-04-23 08:21:38 +0200 (Mo., 23 Apr 2018) $
 *	Last changed by	:	$Author: b7bolm $
 *	URL				:	$URL: http://almscdc.swisslog.com/repo/SWPD/Development/BoxControlFramework/20_Release/trunk/01_Software/BCF/BCF/JumpStart/20_Product/11_Emu/14_Groups/10_Lib/10_Conv/FB_GroupConvEmulation.TcPOU $
 *
 *	Purpose			:	This methode gets always the current values of the real object
 *
 * ------------------------------------------------------------------------------------
 *	Copyright Swisslog [IP AG], Switzerland. All rights reserved.
 * 
 * ------------------------------------------------------------------------------------
 *	
 * 	Revision History: 
 *
 * 	VERSION			DATE			INITIALS			DESCRIPTION
 *	0.1				01.01.2001		swl					Example
 *
 **************************************************************************************)

IF __ISVALIDREF(GroupRegistry[eGroupNumber].rGroupData) THEN
	GroupBase.rGroupDataReal REF= GroupRegistry[eGroupNumber].rGroupData;
ELSE
	GroupBase.rGroupDataReal REF= GroupBase.GroupDataEmpty;
END_IF

IF __ISVALIDREF(GroupRegistry[eGroupNumber].rGroupInterface) THEN
	GroupBase.rGroupInterfaceReal REF= GroupRegistry[eGroupNumber].rGroupInterface;
ELSE
	GroupBase.rGroupInterfaceReal REF= GroupBase.GroupInterfaceEmpty;
END_IF

IF __ISVALIDREF(GroupRegistry[eGroupNumber].rSettingsGroup) THEN
	GroupBase.rSettingsGroupReal REF= GroupRegistry[eGroupNumber].rSettingsGroup;
ELSE
	GroupBase.rSettingsGroupReal REF= GroupBase.SettingsGroupEmpty;
END_IF
END_METHOD

END_FUNCTION_BLOCK

// ---- 20_Product/10_BCF/11_Conv/14_Groups/10_Helper/F_IsGroupInitialized.TcPOU
FUNCTION F_IsGroupInitialized : BOOL
(**************************************************************************************
 * 	Application		:	BoxControl Framework
 *	Revision		:	$Revision: 404529 $
 *	Revision date	:	$Date: 2018-04-23 08:21:38 +0200 (Mo., 23 Apr 2018) $
 *	Last changed by	:	$Author: b7bolm $
 *	URL				:	$URL: http://almscdc.swisslog.com/repo/SWPD/Development/BoxControlFramework/20_Release/trunk/01_Software/BCF/BCF/JumpStart/20_Product/10_App/14_Groups/10_Lib/10_Conv/10_Functions/F_IsGroupInitialized.TcPOU $
 *
 *	Purpose			:	Returns group base data
 *
 * ------------------------------------------------------------------------------------
 *	Copyright Swisslog [IP AG], Switzerland. All rights reserved.
 * 
 * ------------------------------------------------------------------------------------
 *	
 * 	Revision History: 
 *
 * 	VERSION			DATE			INITIALS			DESCRIPTION
 *	0.1				01.01.2001		swl					Example
 *
 **************************************************************************************)
VAR_INPUT
	eGroupNumber		: E_GroupNumber;
END_VAR


// Check if function number is valid
IF eGroupNumber > E_GroupNumber.G_BEGIN_GROUP AND
   eGroupNumber < E_GroupNumber.G_END_GROUP THEN

	// Check reference is valid
	IF __ISVALIDREF(GroupRegistry[eGroupNumber].rGroupData) THEN
   		// Return function data
   		F_IsGroupInitialized := GroupRegistry[eGroupNumber].rGroupData.Init;
	END_IF
END_IF

END_FUNCTION

// ---- 20_Product/10_BCF/11_Conv/14_Groups/10_Helper/F_InitializeGroup.TcPOU
FUNCTION F_InitializeGroup :BOOL
(**************************************************************************************
 * 	Application		:	BoxControl Framework
 *	Revision		:	$Revision: 404529 $
 *	Revision date	:	$Date: 2018-04-23 08:21:38 +0200 (Mo., 23 Apr 2018) $
 *	Last changed by	:	$Author: b7bolm $
 *	URL				:	$URL: http://almscdc.swisslog.com/repo/SWPD/Development/BoxControlFramework/20_Release/trunk/01_Software/BCF/BCF/JumpStart/20_Product/10_App/14_Groups/10_Lib/10_Conv/10_Functions/F_InitializeGroup.TcPOU $
 *
 *	Purpose			:	Initialize group
 *
 * ------------------------------------------------------------------------------------
 *	Copyright Swisslog [IP AG], Switzerland. All rights reserved.
 * 
 * ------------------------------------------------------------------------------------
 *	
 * 	Revision History: 
 *
 * 	VERSION			DATE			INITIALS			DESCRIPTION
 *	0.1				01.01.2001		swl					Example
 *
 **************************************************************************************)
VAR_INPUT
	eGroupNumber		: E_GroupNumber; // Group number
END_VAR


// If reference is valid
IF __ISVALIDREF(GroupRegistry[eGroupNumber].rGroup) THEN
	// Initialize group
	GroupRegistry[eGroupNumber].rGroup.M_InitGroup(TRUE);
END_IF

END_FUNCTION

// ---- 20_Product/20_ProBox/22_ProMove/15_SubSystem/FB_ProBoxSubsystemEmulation.TcPOU
FUNCTION_BLOCK FB_ProBoxSubsystemEmulation EXTENDS FB_SubsystemConvEmulation
VAR
	pSubsystem							: POINTER TO FB_ProBoxSubsystem; // Address to Subsystem
	rSubsystem						: REFERENCE TO FB_ProBoxSubsystem; // Reference to Group
END_VAR


(**************************************************************************************************************
   Initialization
***************************************************************************************************************)
A_Init();


(**************************************************************************************************************
   Update reference
***************************************************************************************************************)
A_UpdateReference();


(**************************************************************************************************************
   Emulation
***************************************************************************************************************)
// If emulation Subsystem is initialized
IF SubsystemData.Init THEN
	// Update real data
	M_UpdateRealObjectData();	

	// Overwrite inputs
	A_OverWriteInputs();
END_IF

ACTION A_Init:
(**************************************************************************************
 * 	NAME		A_Init
 * 	FUNCTION	Initialize emulated Subsystem
 **************************************************************************************)
 
 // If module is not initialized
 IF NOT SubsystemData.Init THEN
	
	IF F_IsSubsystemInitialized() THEN
	
		// Module is initialized
		SubsystemData.Init := TRUE;
	
		// Send debug message
		DebugMsg := CONCAT('Initialization done. Subsystem: ', SubsystemRegistry.SubsystemName);
		fbDebugMsg.M_SendInfoMsg(DebugMsg);		
	
		// Initialize real module
		F_InitializeSubsystem();
	END_IF
END_IF
END_ACTION

ACTION A_OverWriteInputs:
(**************************************************************************************
 * 	NAME		A_OverWriteInputs
 * 	FUNCTION	Overwrite HW-Inputs
 **************************************************************************************)
 
;
END_ACTION

ACTION A_UpdateReference:
(**************************************************************************************
 * 	NAME		A_UpdateReference
 * 	FUNCTION	Update reference to real object
 **************************************************************************************)

// Is reference valid  
IF __ISVALIDREF(SubsystemRegistry.rSubsystem) THEN
	// Build address to reference
	pSubsystem := ADR(SubsystemRegistry.rSubsystem);

	// If address is possible
	IF pSubsystem <> 0 THEN
		// Build reference to memory
		rSubsystem REF= pSubsystem^;
	ELSE
		// Reinitialize module
		SubsystemData.Init := FALSE;
	END_IF
ELSE
	// Reinitialize module
	SubsystemData.Init := FALSE;
END_IF
END_ACTION

END_FUNCTION_BLOCK

// ---- 20_Product/10_BCF/11_Conv/15_Subsystem/09_Emulation/FB_SubsystemConvEmulation.TcPOU
FUNCTION_BLOCK FB_SubsystemConvEmulation EXTENDS FB_BaseObjectEmulation
(**************************************************************************************
 * 	Application		:	BoxControl Framework
 *	Revision		:	$Revision: 404529 $
 *	Revision date	:	$Date: 2018-04-23 08:21:38 +0200 (Mo., 23 Apr 2018) $
 *	Last changed by	:	$Author: b7bolm $
 *	URL				:	$URL: http://almscdc.swisslog.com/repo/SWPD/Development/BoxControlFramework/20_Release/trunk/01_Software/BCF/BCF/JumpStart/20_Product/11_Emu/15_Subsystem/10_Lib/10_Conv/FB_SubsystemConvEmulation.TcPOU $
 *
 *	Purpose			:	Base subsystem - Emulation.
 *
 * ------------------------------------------------------------------------------------
 *	Copyright Swisslog [IP AG], Switzerland. All rights reserved.
 * 
 * ------------------------------------------------------------------------------------
 *	
 * 	Revision History: 
 *
 * 	VERSION			DATE			INITIALS			DESCRIPTION
 *	0.1				01.01.2001		swl					Example
 *
 **************************************************************************************)
VAR
	SubsystemBase					: ST_SubsystemBaseEmulation;
END_VAR

VAR PERSISTENT
	SubsystemData					: ST_SubsystemDataEmulation; // Subsystem data emulation
END_VAR

METHOD PRIVATE M_ITC_ERQ : BOOL
VAR_INPUT
	meChannelSrc		: E_MFCS_CHANNEL; // Number of the source 
	mpData				: PVOID; // Data  pointer 
	mLen				: UDINT; // Data length
END_VAR
// Map data
F_BlockCopy(
	pSrc:= mpData, 
	LenSrc:= mLen, 
	pDest:= ADR(SubsystemBase.ERQ), 
	LenDest:= SIZEOF(SubsystemBase.ERQ));		

// Send "Error" request
SubsystemData.ITC.Commands.Error := SubsystemBase.ERQ.Code = 0;
SubsystemData.ITC.Commands.ErrorCode := SubsystemBase.ERQ.ErrorCode;
END_METHOD

METHOD M_ITC_ProcessMsg : BOOL
VAR_INPUT
	meChannelSrc		: E_MFCS_CHANNEL; // Number of the source 
	mMsgType			: INT; // Message type
	mpData				: PVOID; // Data  pointer 
	mLen				: UDINT; // Data length
END_VAR

// Initialize
M_ITC_ProcessMsg := TRUE;

// Validate inputs
IF mpData > 0 AND
   mLen > 0 THEN
	// Map enum
	SubsystemBase.eITC_MsgType := mMsgType;
	
	// Validate message type
	CASE SubsystemBase.eITC_MsgType OF

		(*******************************************************************************
		  No Message
		********************************************************************************)
		E_ITC_MsgTypeConv.NO_MESSAGE_TYPE:
			// Empty message received
			DebugMsg := 'Empty ITC message received.';
			fbDebugMsg.M_SendErrorMsg(DebugMsg);
			
